{attribute 'global_init_slot' := '40510'}
VAR_GLOBAL
  LblPlt_Facade                                            :FB_BA_Label:=( sObjName:='FAS', sDescr:='Fassade');
  LblPlt_Natural_smoke_extraction                          :FB_BA_Label:=( sObjName:='NRA', sDescr:='Natürlicher Rauchabzug');
  LblPlt_Doors_gates_sluices                               :FB_BA_Label:=( sObjName:='TUE', sDescr:='Türen, Tore, Schleusen');
  LblPlt_Smoke_and_heat_extraction_system                  :FB_BA_Label:=( sObjName:='RWA', sDescr:='Rauch- und Wärmeabzugsanlage');
  LblPlt_Sunlight_protection                               :FB_BA_Label:=( sObjName:='SON', sDescr:='Sonnenschutzanlage');
// 411 Abwasseranlagen
  LblPlt_Separator_facility                                :FB_BA_Label:=( sObjName:='ABS', sDescr:='Abscheideranlage');
  LblPlt_Lifting_system                                    :FB_BA_Label:=( sObjName:='HBA', sDescr:='Hebeanlage');
  LblPlt_Neutralisation_plant                              :FB_BA_Label:=( sObjName:='NEU', sDescr:='Neutralisationsanlage');
// 412 Wasseranlagen
  LblPlt_Trace_heating                                     :FB_BA_Label:=( sObjName:='BGH', sDescr:='Begleitheizung');
  LblPlt_Process_water                                     :FB_BA_Label:=( sObjName:='BTW', sDescr:='Betriebswasser');
  LblPlt_Well_water                                        :FB_BA_Label:=( sObjName:='BWA', sDescr:='Brunnenwasser');
  LblPlt_Dispensing_installation                           :FB_BA_Label:=( sObjName:='DOS', sDescr:='Dosieranlage');
  LblPlt_Pressure_booster_system                           :FB_BA_Label:=( sObjName:='DEA', sDescr:='Druckerhöhungsanlage');
  LblPlt_Softening_unit                                    :FB_BA_Label:=( sObjName:='EHA', sDescr:='Enthärtungsanlage');
// Trinkwasser
  LblPlt_Drinking_water_heating_system                     :FB_BA_Label:=( sObjName:='TWE', sDescr:='Trinkwassererwärmungsanlage');
  LblPlt_Reverse_osmosis_system                            :FB_BA_Label:=( sObjName:='UKO', sDescr:='Umkehrosmoseanlage');
  LblPlt_Desalination_plant                                :FB_BA_Label:=( sObjName:='VEA', sDescr:='Vollentsalzungsanlage');
// 421 Wärmeerzeugungsanlagen
  LblPlt_BHKW                                              :FB_BA_Label:=( sObjName:='BHK', sDescr:='BHKW');
  LblPlt_Electric_heating                                  :FB_BA_Label:=( sObjName:='EHZ', sDescr:='Elektroheizung');
  LblPlt_District_heating_transfer                         :FB_BA_Label:=( sObjName:='FWÜ', sDescr:='Fernwärmeübergabe');
// Geothermieanlage
  LblPlt_Boiler                                            :FB_BA_Label:=( sObjName:='KES', sDescr:='Kessel');
  LblPlt_Clean_steam_generation                            :FB_BA_Label:=( sObjName:='RDE', sDescr:='Reindampferzeugung');
  LblPlt_Solar_power_system                                :FB_BA_Label:=( sObjName:='SOL', sDescr:='Solaranlage');
  LblPlt_Heating_pump                                      :FB_BA_Label:=( sObjName:='WPU', sDescr:='Wärmepumpe');
// 422 Wärmeverteilnetze
  LblPlt_Pressure_maintenance                              :FB_BA_Label:=( sObjName:='DHG', sDescr:='Druckhaltung');
  LblPlt_Heating_circuit                                   :FB_BA_Label:=( sObjName:='HZK', sDescr:='Heizkreis');
  LblPlt_Heating                                           :FB_BA_Label:=( sObjName:='HZG', sDescr:='Heizung');
  LblPlt_Back_feed_system                                  :FB_BA_Label:=( sObjName:='NSA', sDescr:='Nachspeiseanlage');
  LblPlt_Buffer                                            :FB_BA_Label:=( sObjName:='PFS', sDescr:='Pufferspeicher');
  LblPlt_Heat_distribution_network                         :FB_BA_Label:=( sObjName:='WVN', sDescr:='Wärmeverteilnetz');
  LblPlt_Heat_exchanger                                    :FB_BA_Label:=( sObjName:='WTR', sDescr:='Wärmeüberträger');
// 423 Raumheizflächen
  LblPlt_Concrete_core_activation                          :FB_BA_Label:=( sObjName:='BKA', sDescr:='Betonkernaktivierung');
  LblPlt_Overhead_heating                                  :FB_BA_Label:=( sObjName:='DHZ', sDescr:='Deckenheizung');
  LblPlt_Ceiling_radiator_panels                           :FB_BA_Label:=( sObjName:='DSP', sDescr:='Deckenstrahlplatten');
  LblPlt_Facade_heating                                    :FB_BA_Label:=( sObjName:='FAH', sDescr:='Fassadenheizung');
  LblPlt_Panel_heating                                     :FB_BA_Label:=( sObjName:='FLH', sDescr:='Flächenheizung');
  LblPlt_Underfloor_heating                                :FB_BA_Label:=( sObjName:='FBH', sDescr:='Fußbodenheizung');
  LblPlt_Heated_chilled_ceiling                            :FB_BA_Label:=( sObjName:='HKD', sDescr:='Heiz-/Kühldecke');
  LblPlt_Static_heating                                    :FB_BA_Label:=( sObjName:='STH', sDescr:='Statische Heizung');
// 430 Lufttechnische Anlagen
  LblPlt_Extract_air_system                                :FB_BA_Label:=( sObjName:='ABA', sDescr:='Abluftanlage');
  LblPlt_Roof_air_heater                                   :FB_BA_Label:=( sObjName:='DLH', sDescr:='Deckenlufterhitzer');
  LblPlt_Circulatory_system                                :FB_BA_Label:=( sObjName:='KVS', sDescr:='Kreislaufverbundsystem');
  LblPlt_Air_processing_unit                               :FB_BA_Label:=( sObjName:='LAZ', sDescr:='Luftaufbereitungszentrale');
  LblPlt_Mechanical_smoke_extraction_system                :FB_BA_Label:=( sObjName:='MRA', sDescr:='Maschinelle Rauchabzugsanlage');
  LblPlt_Smoke_pressure_system                             :FB_BA_Label:=( sObjName:='RDA', sDescr:='Rauchdruckanlage');
  LblPlt_Air_handling_unit                                 :FB_BA_Label:=( sObjName:='RLT', sDescr:='Raumlufttechnik');
  LblPlt_Partial_air_conditioning_system                   :FB_BA_Label:=( sObjName:='TKA', sDescr:='Teilklimaanlage');
  LblPlt_Air_curtain_system                                :FB_BA_Label:=( sObjName:='TLS', sDescr:='Türluftschleieranlage');
  LblPlt_Recirculating_air_system                          :FB_BA_Label:=( sObjName:='ULA', sDescr:='Umluftanlage');
  LblPlt_Full_air_conditioning_system                      :FB_BA_Label:=( sObjName:='VKA', sDescr:='Vollklimaanlage');
  LblPlt_Heat_recovery_system                              :FB_BA_Label:=( sObjName:='WRG', sDescr:='Wärmerückgewinnungssystem');
  LblPlt_Intake_air_system                                 :FB_BA_Label:=( sObjName:='ZUA', sDescr:='Zuluftanlage');
  LblPlt_Smoke_extraction_system                           :FB_BA_Label:=( sObjName:='ERA', sDescr:='Entrauchungsanlage');
// 434 Kälteanlagen
  LblPlt_Remote_cooling_transfer                           :FB_BA_Label:=( sObjName:='FKÜ', sDescr:='Fernkälteübergabe');
  LblPlt_Cooling                                           :FB_BA_Label:=( sObjName:='KAE', sDescr:='Kälte');
  LblPlt_Cooling_circuit                                   :FB_BA_Label:=( sObjName:='KKR', sDescr:='Kältekreis');
  LblPlt_Cooling_distribution_network                      :FB_BA_Label:=( sObjName:='KVN', sDescr:='Kälteverteilnetz');
  LblPlt_Cold_water_generation                             :FB_BA_Label:=( sObjName:='KWE', sDescr:='Kaltwassererzeugung');
  LblPlt_Electrical_cabinet_cooling                        :FB_BA_Label:=( sObjName:='KVE', sDescr:='Kühlung Schaltschrank ');
  LblPlt_Cooling_storage                                   :FB_BA_Label:=( sObjName:='KSP', sDescr:='Kältespeicher');
  LblPlt_Chilled_ceiling                                   :FB_BA_Label:=( sObjName:='KÜD', sDescr:='Kühldecke');
  LblPlt_Re_cooling_plant                                  :FB_BA_Label:=( sObjName:='RKW', sDescr:='Rückkühlwerk');
// 441 Hoch- und Mittelspannungsanlagen
  LblPlt_Switchgear                                        :FB_BA_Label:=( sObjName:='STA', sDescr:='Schaltanlagen');
  LblPlt_Transformer                                       :FB_BA_Label:=( sObjName:='TRF', sDescr:='Transformator');
  LblPlt_Medium_voltage_system                             :FB_BA_Label:=( sObjName:='MSA', sDescr:='Mittelspannungsanlage');
  LblPlt_Compensation_system                               :FB_BA_Label:=( sObjName:='KOA', sDescr:='Kompensationsanlage');
  LblPlt_Frequency_converter_system                        :FB_BA_Label:=( sObjName:='FUA', sDescr:='Frequenzumformeranlage');
// 442 Eigenstromversorgungsanlagen
  LblPlt_Emissions_system                                  :FB_BA_Label:=( sObjName:='AGA', sDescr:='Abgasanlage');
  LblPlt_Battery_unit                                      :FB_BA_Label:=( sObjName:='BAT', sDescr:='Batterieanlage');
  LblPlt_Co_generation_unit                                :FB_BA_Label:=( sObjName:='BHK', sDescr:='Blockheizkraftwerk');
  LblPlt_Fuel_supply                                       :FB_BA_Label:=( sObjName:='BRV', sDescr:='Brennstoffversorgung');
  LblPlt_Standby_power_system                              :FB_BA_Label:=( sObjName:='ESA', sDescr:='Ersatzstromanlage');
  LblPlt_Photovoltaic_system                               :FB_BA_Label:=( sObjName:='PVA', sDescr:='Fotovoltaikanlage');
  LblPlt_Uninterruptible_power_supply                      :FB_BA_Label:=( sObjName:='USV', sDescr:='Unterbrechungsfreie Stromversorgung');
// 443 Niederspannungsschaltanlagen
  LblPlt_General_power_supply                              :FB_BA_Label:=( sObjName:='ASV', sDescr:='Allgemeine Stromversorgung');
  LblPlt_Safety_power_supply                               :FB_BA_Label:=( sObjName:='SSV', sDescr:='Sicherheitsstromversorgung');
  LblPlt_Lighting                                          :FB_BA_Label:=( sObjName:='BEL', sDescr:='Beleuchtungsanlage');
  LblPlt_Emergency_lighting                                :FB_BA_Label:=( sObjName:='SIB', sDescr:='Sicherheitsbeleuchtung');
// 451 Telekommunikationsanlagen
  LblPlt_Telecommunications_system                         :FB_BA_Label:=( sObjName:='TEL', sDescr:='Telekommunikationsanlage');
// 452 Such- und Signalanlagen
  LblPlt_Call_signalling_system                            :FB_BA_Label:=( sObjName:='LRA', sDescr:='Lichtrufanlage');
  LblPlt_Door_intercom_and_door_opener_system              :FB_BA_Label:=( sObjName:='TÜA', sDescr:='Türsprech- und -öffneranlage');
  LblPlt_Paging_system                                     :FB_BA_Label:=( sObjName:='PRA', sDescr:='Personenrufanlage');
// 453 Zeitdienstanlagen
  LblPlt_Clock_and_time_recording_system                   :FB_BA_Label:=( sObjName:='ZEA', sDescr:='Uhren- und Zeiterfassungsanlage');
// 454 Elektroakustische Anlagen
  LblPlt_Electro_acoustic_sound_systems                    :FB_BA_Label:=( sObjName:='ELA', sDescr:='Elektroakustische Anl. , Beschallung');
  LblPlt_Conference_and_interpreting_equipment             :FB_BA_Label:=( sObjName:='KDA', sDescr:='Konferenz- und Dolmetscheranlage');
  LblPlt_Intercom_system                                   :FB_BA_Label:=( sObjName:='GSA', sDescr:='Gegensprechanlage');
  LblPlt_Voice_alarm_system                                :FB_BA_Label:=( sObjName:='SAA', sDescr:='Sprachalarmierungsanlage');
  LblPlt_Intercommunication_systems                        :FB_BA_Label:=( sObjName:='WSA', sDescr:='Wechselsprechanlagen');
// 455 Fernseh- und Antennenanlagen
  LblPlt_Television_system                                 :FB_BA_Label:=( sObjName:='TVA', sDescr:='Fernsehanlage');
  LblPlt_Transmitting_and_receiving_antenna_system         :FB_BA_Label:=( sObjName:='SEA', sDescr:='Sende- und Empfangsantennenanlage');
  LblPlt_BOS_radio_system                                  :FB_BA_Label:=( sObjName:='BOS', sDescr:='BOS-Funkanlage');
// 456 Gefahrenmelde- und Alarmanlagen
  LblPlt_Fire_detection_and_alarm_systems                  :FB_BA_Label:=( sObjName:='BMA', sDescr:='Brandmeldeanlage');
  LblPlt_Carbon_monoxide_warning_system                    :FB_BA_Label:=( sObjName:='COW', sDescr:='CO-Warnanlage');
  LblPlt_Burglar_alarm_systems                             :FB_BA_Label:=( sObjName:='EMA', sDescr:='Einbruchmeldeanlage');
  LblPlt_Fire_control_panel                                :FB_BA_Label:=( sObjName:='FWT', sDescr:='Feuerwehrtableau');
  LblPlt_Escape_route_protection_system                    :FB_BA_Label:=( sObjName:='FWS', sDescr:='Fluchtwegsicherungsanlage');
  LblPlt_Hazard_detection_system                           :FB_BA_Label:=( sObjName:='GMA', sDescr:='Gefahrenmeldeanlage');
  LblPlt_Gas_warning_system                                :FB_BA_Label:=( sObjName:='GWA', sDescr:='Gaswarnanlage');
  LblPlt_Smoke_aspiration_system                           :FB_BA_Label:=( sObjName:='RAS', sDescr:='Rauchansaugsystem');
  LblPlt_Room_observation_system                           :FB_BA_Label:=( sObjName:='RBA', sDescr:='Raumbeobachtungsanlage');
  LblPlt_Robbery_alarm_system                              :FB_BA_Label:=( sObjName:='ÜFA', sDescr:='Überfallmeldeanlage');
  LblPlt_Guard_control_system                              :FB_BA_Label:=( sObjName:='WKA', sDescr:='Wächterkontrollanlage');
  LblPlt_Emergency_call_system                             :FB_BA_Label:=( sObjName:='NOT', sDescr:='Notrufanlage');
  LblPlt_Access_control_system                             :FB_BA_Label:=( sObjName:='ZKS', sDescr:='Zugangskontrollsystem');
// 457 Übertragungsnetze
  LblPlt_Networks_for_the_transmission_voice_text_etc      :FB_BA_Label:=( sObjName:='LAN', sDescr:='Netzw.  Daten, Sprache, Text etc');
// 459 Fernmelde- und informationstechnische Anlagen, Sonstiges
  LblPlt_Remote_control_systems                            :FB_BA_Label:=( sObjName:='FWA', sDescr:='Fernwirkanlagen');
  LblPlt_Parking_guidance_systems                          :FB_BA_Label:=( sObjName:='PLS', sDescr:='Parkleitsysteme');
// 460 Förderanlagen
  LblPlt_File_transportation_systems                       :FB_BA_Label:=( sObjName:='ATA', sDescr:='Aktentransportanlagen');
  LblPlt_Lift                                              :FB_BA_Label:=( sObjName:='AUF', sDescr:='Aufzug');
  LblPlt_Inspection_systems                                :FB_BA_Label:=( sObjName:='BFA', sDescr:='Befahranlagen');
  LblPlt_Moving_walkways                                   :FB_BA_Label:=( sObjName:='FST', sDescr:='Fahrsteige');
  LblPlt_Escalators                                        :FB_BA_Label:=( sObjName:='FTR', sDescr:='Fahrtreppen');
  LblPlt_External_lifts                                    :FB_BA_Label:=( sObjName:='FSA', sDescr:='Fassadenaufzüge');
  LblPlt_Baggage_conveyor_system                           :FB_BA_Label:=( sObjName:='GFA', sDescr:='Gepäckförderanlage');
  LblPlt_Pneumatic_delivery_systems                        :FB_BA_Label:=( sObjName:='RPA', sDescr:='Rohrpostanlagen');
  LblPlt_Goods_transportation_facilities                   :FB_BA_Label:=( sObjName:='WTA', sDescr:='Warentransportanlagen');
// 470 Nutzerspezifische Anlagen
// 471 Küchentechnische Anlagen
  LblPlt_Small_refrigeration_unit                          :FB_BA_Label:=( sObjName:='KLK', sDescr:='Kleinkälteanlage');
// 472 Wäscherei- und Reinigungsanlagen
  LblPlt_Disinfection_unit                                 :FB_BA_Label:=( sObjName:='DES', sDescr:='Desinfektionsanlage');
  LblPlt_Cleaning_unit                                     :FB_BA_Label:=( sObjName:='REA', sDescr:='Reinigungsanlage');
  LblPlt_Sterilisation_systems                             :FB_BA_Label:=( sObjName:='STR', sDescr:='Sterilisationseinrichtungen');
  LblPlt_Water_treatment_system                            :FB_BA_Label:=( sObjName:='WAA', sDescr:='Wasseraufbereitungsanlage');
  LblPlt_Laundry_system                                    :FB_BA_Label:=( sObjName:='WÄA', sDescr:='Wäschereianlage');
// 473 Medienversorgungsanlagen
  LblPlt_Compressed_air_supply_system                      :FB_BA_Label:=( sObjName:='DRL', sDescr:='Druckluftversorgungsanlage');
  LblPlt_Pressure_regulator_unit                           :FB_BA_Label:=( sObjName:='DRA', sDescr:='Druckregelanlage');
  LblPlt_Media_supply_system                               :FB_BA_Label:=( sObjName:='MVA', sDescr:='Medienversorgungsanlage');
  LblPlt_Medical_and_technical_gases                       :FB_BA_Label:=( sObjName:='MTG', sDescr:='Medizinische und technische Gase');
  LblPlt_Vacuum_unit                                       :FB_BA_Label:=( sObjName:='VAK', sDescr:='Vakuumanlage');
// 474 Medizin- und labortechnische Anlagen
  LblPlt_Medical_technical_plant                           :FB_BA_Label:=( sObjName:='MED', sDescr:='Medizintechnische Anlagen');
  LblPlt_Medical_gas_supply                                :FB_BA_Label:=( sObjName:='MGV', sDescr:='Medizinische Gasversorgung');
  LblPlt_Laboratory_equipment                              :FB_BA_Label:=( sObjName:='LAB', sDescr:='Labortechnische Anlagen (allgemein)');
// 475 Feuerlöschanlagen
  LblPlt_Fire_extinguisher                                 :FB_BA_Label:=( sObjName:='FLA', sDescr:='Feuerlöschanlage');
  LblPlt_Gas_extinguishing_system                          :FB_BA_Label:=( sObjName:='GLA', sDescr:='Gaslöschanlage');
  LblPlt_Fire_extinguishing_system                         :FB_BA_Label:=( sObjName:='LÖS', sDescr:='Löschanlage (allgemein)');
  LblPlt_Mist_extinguishing_system                         :FB_BA_Label:=( sObjName:='NLA', sDescr:='Nebellöschanlage');
  LblPlt_NOX_system                                        :FB_BA_Label:=( sObjName:='NOX', sDescr:='NOX-Anlage');
  LblPlt_Sprinkler_system                                  :FB_BA_Label:=( sObjName:='SPR', sDescr:='Sprinkleranlage');
  LblPlt_Wall_hydrant_system                               :FB_BA_Label:=( sObjName:='WHA', sDescr:='Wandhydrantenanlage');
// 478 Entsorgungsanlagen
  LblPlt_Waste_disposal_system                             :FB_BA_Label:=( sObjName:='AEA', sDescr:='Abfallentsorgungsanlage');
  LblPlt_Media_disposal_system                             :FB_BA_Label:=( sObjName:='MEA', sDescr:='Medienentsorgungsanlage');
  LblPlt_Vacuum_cleaning_systems                           :FB_BA_Label:=( sObjName:='SSA', sDescr:='Staubsauganlagen');
// 480 Gebäudeautomation
  LblPlt_Automation_control_equipment                      :FB_BA_Label:=( sObjName:='ASP', sDescr:='Automationsschwerpunkt');
  LblPlt_Weather_station                                   :FB_BA_Label:=( sObjName:='WET', sDescr:='Wetterstation');
  LblPlt_Weather_data                                      :FB_BA_Label:=( sObjName:='WED', sDescr:='Wetterdaten');
  LblPlt_Management_and_operating_equipment                :FB_BA_Label:=( sObjName:='MBE', sDescr:='Management- und Bedieneinrichtungen');
  LblPlt_Room_automation                                   :FB_BA_Label:=( sObjName:='RAU', sDescr:='Raumautomation');
  LblPlt_Room_automation_system_distributor                :FB_BA_Label:=( sObjName:='RAV', sDescr:='Raumautomation-Systemverteiler');
  LblPlt_Control_cabinet                                   :FB_BA_Label:=( sObjName:='SSK', sDescr:='Schaltschrank');
  LblPlt_Settings                                          :FB_BA_Label:=( sObjName:='ALP', sDescr:='Anlagenparameter');
  LblPlt_EventGroups                                       :FB_BA_Label:=( sObjName:='ERG', sDescr:='Meldeklassen');
  LblPlt_Global_building_data                              :FB_BA_Label:=( sObjName:='GGL', sDescr:='Globale Gebäudedaten');
// 540 Technische Anlagen in Außenanlagen
  LblPlt_Rainwater_retention_basin                         :FB_BA_Label:=( sObjName:='RRB', sDescr:='Regenrückhaltebecken');
  LblPlt_Cistern_system                                    :FB_BA_Label:=( sObjName:='ZTA', sDescr:='Zisternenanlage');
END_VAR

// ---- Templates/GVLs/Language/German/TxtEvent_DE.TcGVL
{region '#Template'}
	{attribute 'Version' := '5.1.0.0'}
	{attribute 'Tags' := '"LCID": "1031", "Text": "GVL, Property, Event, Event Message Text, Active Text, Inactive Text"'}
	{attribute 'Tags' := '"LCID": "1033", "Text": "GVL, Property, Event, Event Message Text, Active Text, Inactive Text"'}
	{attribute 'Description' := '"LCID": "1031", "Text": "Textliste Properties Event Message Text, Active Text, Inactive Text"'}
	{attribute 'Description' := '"LCID": "1033", "Text": "Text list Properties Event Message Text, Active Text, Inactive Text"'}
{endregion}

{attribute 'global_init_slot' := '40510'}
VAR_GLOBAL
  txtEvent_No                                                :T_BA_StateText:='Nein';
  txtEvent_Yes                                               :T_BA_StateText:='Ja';
  txtEvent_Auto                                              :T_BA_StateText:='Automatik';
  txtEvent_Manual                                            :T_BA_StateText:='Hand';
  txtEvent_Off                                               :T_BA_StateText:='Aus';
  txtEvent_On                                                :T_BA_StateText:='Ein';
  txtEvent_Opened                                            :T_BA_StateText:='Geöffnet';
  txtEvent_Closed                                            :T_BA_StateText:='Geschlossen';
  txtEvent_Open                                              :T_BA_StateText:='Auf';
  txtEvent_Close                                             :T_BA_StateText:='Zu';
  txtEvent_Step1                                             :T_BA_StateText:='Stufe 1 ';
  txtEvent_Step2                                             :T_BA_StateText:='Stufe 2';
  txtEvent_Step3                                             :T_BA_StateText:='Stufe 3';
  txtEvent_Step4                                             :T_BA_StateText:='Stufe 4';
  txtEvent_Step5                                             :T_BA_StateText:='Stufe 5';
  txtEvent_Step6                                             :T_BA_StateText:='Stufe 6';
  txtEvent_Step7                                             :T_BA_StateText:='Stufe 7';
  txtEvent_Step8                                             :T_BA_StateText:='Stufe 8';
  txtEvent_Released                                          :T_BA_StateText:='Freigegeben';
  txtEvent_Inactive                                          :T_BA_StateText:='Inaktiv';
  txtEvent_Active                                            :T_BA_StateText:='Aktiv';
  txtEvent_Normal                                            :T_BA_StateText:='Normal';
  txtEvent_Offnormal                                         :T_BA_StateText:='Unnormal';
  txtEvent_Alert                                             :T_BA_StateText:='Alarm';
  txtEvent_Disturb                                           :T_BA_StateText:='Störung';
  txtEvent_Error                                             :T_BA_StateText:='Fehler ';
  txtEvent_Triggered                                         :T_BA_StateText:='Ausgelöst';
  txtEvent_Maintenace                                        :T_BA_StateText:='Wartung';
  txtEvent_Exceeded                                          :T_BA_StateText:='Überschritten';
  txtEvent_Monitoring                                        :T_BA_StateText:='Überwachung';
  txtEvent_Protection                                        :T_BA_StateText:='Schutzbetrieb';
  txtEvent_Economy                                           :T_BA_StateText:='Economy';
  txtEvent_PreComfort                                        :T_BA_StateText:='Pre-Comfort';
  txtEvent_Comfort                                           :T_BA_StateText:='Comfort';
  txtEvent_Reached                                           :T_BA_StateText:='erreicht';
  txtEvent_NotReached                                        :T_BA_StateText:='nicht erreicht';
  txtEvent_None                                              :T_BA_StateText:='""';
  txtEvent_EmergencyStop                                     :T_BA_StateText:='Notaus';
  txtEvent_Frost                                             :T_BA_StateText:='Frost';
  txtEvent_SmokeExtraction_P                                 :T_BA_StateText:='Entrauchung mit Zu- und Abluft';
  txtEvent_SmokeExtractionSupplyAir                          :T_BA_StateText:='Entrauchung Zuluft';
  txtEvent_SmokeExtractionExtractAir                         :T_BA_StateText:='Entrauchung Abluft';
  txtEvent_CoolDownProtection                                :T_BA_StateText:='Auskühlschutz';
  txtEvent_OverHeatingProtection                             :T_BA_StateText:='Überhitzungsschutz';
  txtEvent_Fire                                              :T_BA_StateText:='Brandalarm';
  txtEvent_NightCooling                                      :T_BA_StateText:='Nachtkühlung';
  txtEvent_ForcedVentilation                                 :T_BA_StateText:='Zwangsbelüftung';
  txtEvent_CentralSwitchOff                                  :T_BA_StateText:='Zentralaus';
  txtEvent_Locked                                            :T_BA_StateText:='verriegelt';
  txtEvent_Contaminated                                      :T_BA_StateText:='verschmutzt';
  txtEvent_Stop                                              :T_BA_StateText:='Stop';
  txtEvent_Critical                                          :T_BA_StateText:='kritisch';
  txtEvent_CriticalOn                                        :T_BA_StateText:='kritisch ein';
  txtEvent_CriticalOff                                       :T_BA_StateText:='kritisch aus';
  txtEvent_UnCiritical                                       :T_BA_StateText:='unkritisch';
  txtEvent_LifeSafetyOn                                      :T_BA_StateText:='Lebensgefahr ein';
  txtEvent_LifeSafetyOff                                     :T_BA_StateText:='Lebensgefahr aus';
  txtEvent_Average                                           :T_BA_StateText:='Mittelwert';
  txtEvent_HeatCool                                          :T_BA_StateText:='Heiz/Kühl';
  txtEvent_AverageHeatCool                                   :T_BA_StateText:='Mittelwert Heizen/Kühlen';
  txtEvent_Direction                                         :T_BA_StateText:='Wirksinn';
  txtEvent_Default                                           :T_BA_StateText:='Standard';
  txtEvent_Cleaning                                          :T_BA_StateText:='Gebaeudereinigung';
  txtEvent_Nightwatch                                        :T_BA_StateText:='Nachtwaechter';
  txtEvent_SupplyAirTControlReheater                         :T_BA_StateText:='Zulufttemperaturregelung Nacherhitzer';
  txtEvent_SupplyAirTControlPreheater                        :T_BA_StateText:='Zulufttemperaturregelung Vorerhitzer';
  txtEvent_SupplyAirTControlERC                              :T_BA_StateText:='Zulufttemperaturregelung WRG';
  txtEvent_SupplyAirTControlMix                              :T_BA_StateText:='Zulufttemperaturregelung Mischluft';
  txtEvent_SupplyAirTControlCooler                           :T_BA_StateText:='Zulufttemperaturregelung Kühler';
  txtEvent_SupplyAirXControlCooler                           :T_BA_StateText:='Zuluftfeuchtereglung Kühler';
  txtEvent_SupplyAirXControlHumf                             :T_BA_StateText:='Zuluftfeuchtereglung Befeuchter';
  txtEvent_PreRinse                                          :T_BA_StateText:='Vorspülen';
  txtEvent_DamperOpen                                        :T_BA_StateText:='Klappen Auf';
  txtEvent_SupplyAirFan                                      :T_BA_StateText:='Zuluft Ventilator';
  txtEvent_ExtractAirFan                                     :T_BA_StateText:='Abluft Ventilator';
  txtEvent_EnableTemperatureControl                          :T_BA_StateText:='Freigabe Temperatur Regelung';
  txtEvent_EnableTemperatureSequenceLink                     :T_BA_StateText:='Freigabe Temperatur Sequenz Steuerung';
  txtEvent_EnableHumidityControl                             :T_BA_StateText:='Freigabe Feuchte Regelung';
  txtEvent_EnableHumiditySequenceLink                        :T_BA_StateText:='Freigabe Feuchte Sequenz Steuerung';
  txtEvent_ReleaseLimitMonitoring                            :T_BA_StateText:='Freigabe Grenzwertüberwachung';
  txtEvent_Reheater                                          :T_BA_StateText:='Nacherhitzer';
  txtEvent_Preheater                                         :T_BA_StateText:='Vorerhitzer';
  txtEvent_MixedAir                                          :T_BA_StateText:='Mischluft';
  txtEvent_EnergyRecovery                                    :T_BA_StateText:='Energierückgewinnung';
  txtEvent_Cooler                                            :T_BA_StateText:='Kühler';
  txtEvent_Humidifier                                        :T_BA_StateText:='Befeuchter';
  txtEvent_Dehumidifier                                      :T_BA_StateText:='Entfeuchter';
  txtEvent_DamperExhaustAir                                  :T_BA_StateText:='Fortluftklappe';
  txtEvent_DamperOutsideAir                                  :T_BA_StateText:='Aussenluftklappe';
  txtEvent_Occupied                                          :T_BA_StateText:='Belegt';
  txtEvent_NotOccupied                                       :T_BA_StateText:='Nicht belegt';
  txtEvent_Storm                                             :T_BA_StateText:='Sturmalarm';
  txtEvent_Ice                                               :T_BA_StateText:='Vereisung';
  txtEvent_CommError                                         :T_BA_StateText:='Kommunikationsfehler';
  txtEvent_Burglary                                          :T_BA_StateText:='Einbruch';
  txtEvent_Maintenance                                       :T_BA_StateText:='Wartung';
  txtEvent_Referencing                                       :T_BA_StateText:='Referenzieren';
  txtEvent_ManualActuator                                    :T_BA_StateText:='Hand Einzel';
  txtEvent_ManualGroup                                       :T_BA_StateText:='Hand Gruppe';
  txtEvent_AllDown                                           :T_BA_StateText:='Alle herab';
  txtEvent_AllUp                                             :T_BA_StateText:='Alle herauf';
  txtEvent_Scene1                                            :T_BA_StateText:='Szene 1';
  txtEvent_FacadeThermoAutomatic                             :T_BA_StateText:='Fassaden-Thermoautomatik';
  txtEvent_FacadeTwilightAutomatic                           :T_BA_StateText:='Fassaden-Dämmerungsautomatik';
  txtEvent_ParkPosition                                      :T_BA_StateText:='Parkposition';
  txtEvent_Scene2                                            :T_BA_StateText:='Szene 2';
  txtEvent_Scene3                                            :T_BA_StateText:='Szene 3';
  txtEvent_SunProtection                                     :T_BA_StateText:='Sonnenschutz';
  txtEvent_GroupThermoAuto                                   :T_BA_StateText:='Thermoautomatik';
  txtEvent_GroupTwiLightAuto                                 :T_BA_StateText:='Dämmerungsautomatik';
  txtEvent_UserDefined1                                      :T_BA_StateText:='Benutzerdefiniert 1';
  txtEvent_UserDefined2                                      :T_BA_StateText:='Benutzerdefiniert 2';
END_VAR

// ---- Templates/GVLs/Language/German/TxtPlant_DE.TcGVL
{region '#Template'}
	{attribute 'Version' := '5.0.0.0'}
	{attribute 'Tags' := '"LCID": "1031", "Text": "GVL, DPAD, Plants, ObjectName, Description"'}
	{attribute 'Tags' := '"LCID": "1033", "Text": "GVL, DPAD, Plants, ObjectName, Description"'}
	{attribute 'Description' := '"LCID": "1031", "Text": "Textliste Anlagen"'}
	{attribute 'Description' := '"LCID": "1033", "Text": "Text list plants"'}
{endregion}

{attribute 'global_init_slot' := '40510'}
VAR_GLOBAL
  TxTPlant_Facade_sObjectName                                            :T_BA_StateText:='FAS';
  TxTPlant_Facade_sDescription                                            :T_BA_StateText:='Fassade';
  TxTPlant_Natural_smoke_extraction_sObjectName                          :T_BA_StateText:='NRA';
  TxTPlant_Natural_smoke_extraction_sDescription                          :T_BA_StateText:='Natürlicher Rauchabzug';
  TxTPlant_Doors_gates_sluices_sObjectName                               :T_BA_StateText:='TUE';
  TxTPlant_Doors_gates_sluices_sDescription                               :T_BA_StateText:='Türen, Tore, Schleusen';
  TxTPlant_Smoke_and_heat_extraction_system_sObjectName                  :T_BA_StateText:='RWA';
  TxTPlant_Smoke_and_heat_extraction_system_sDescription                  :T_BA_StateText:='Rauch- und Wärmeabzugsanlage';
  TxTPlant_Sunlight_protection_sObjectName                               :T_BA_StateText:='SON';
  TxTPlant_Sunlight_protection_sDescription                               :T_BA_StateText:='Sonnenschutzanlage';
// 411 Abwasseranlagen
  TxTPlant_Separator_facility_sObjectName                                :T_BA_StateText:='ABS';
  TxTPlant_Separator_facility_sDescription                                :T_BA_StateText:='Abscheideranlage';
  TxTPlant_Lifting_system_sObjectName                                    :T_BA_StateText:='HBA';
  TxTPlant_Lifting_system_sDescription                                    :T_BA_StateText:='Hebeanlage';
  TxTPlant_Neutralisation_plant_sObjectName                              :T_BA_StateText:='NEU';
  TxTPlant_Neutralisation_plant_sDescription                              :T_BA_StateText:='Neutralisationsanlage';
// 412 Wasseranlagen
  TxTPlant_Trace_heating_sObjectName                                     :T_BA_StateText:='BGH';
  TxTPlant_Trace_heating_sDescription                                     :T_BA_StateText:='Begleitheizung';
  TxTPlant_Process_water_sObjectName                                     :T_BA_StateText:='BTW';
  TxTPlant_Process_water_sDescription                                     :T_BA_StateText:='Betriebswasser';
  TxTPlant_Well_water_sObjectName                                        :T_BA_StateText:='BWA';
  TxTPlant_Well_water_sDescription                                        :T_BA_StateText:='Brunnenwasser';
  TxTPlant_Dispensing_installation_sObjectName                           :T_BA_StateText:='DOS';
  TxTPlant_Dispensing_installation_sDescription                           :T_BA_StateText:='Dosieranlage';
  TxTPlant_Pressure_booster_system_sObjectName                           :T_BA_StateText:='DEA';
  TxTPlant_Pressure_booster_system_sDescription                           :T_BA_StateText:='Druckerhöhungsanlage';
  TxTPlant_Softening_unit_sObjectName                                    :T_BA_StateText:='EHA';
  TxTPlant_Softening_unit_sDescription                                    :T_BA_StateText:='Enthärtungsanlage';
// Trinkwasser
  TxTPlant_Drinking_water_heating_system_sObjectName                     :T_BA_StateText:='TWE';
  TxTPlant_Drinking_water_heating_system_sDescription                     :T_BA_StateText:='Trinkwassererwärmungsanlage';
  TxTPlant_Reverse_osmosis_system_sObjectName                            :T_BA_StateText:='UKO';
  TxTPlant_Reverse_osmosis_system_sDescription                            :T_BA_StateText:='Umkehrosmoseanlage';
  TxTPlant_Desalination_plant_sObjectName                                :T_BA_StateText:='VEA';
  TxTPlant_Desalination_plant_sDescription                                :T_BA_StateText:='Vollentsalzungsanlage';
// 421 Wärmeerzeugungsanlagen
  TxTPlant_BHKW_sObjectName                                              :T_BA_StateText:='BHK';
  TxTPlant_BHKW_sDescription                                              :T_BA_StateText:='BHKW';
  TxTPlant_Electric_heating_sObjectName                                  :T_BA_StateText:='EHZ';
  TxTPlant_Electric_heating_sDescription                                  :T_BA_StateText:='Elektroheizung';
  TxTPlant_District_heating_transfer_sObjectName                         :T_BA_StateText:='FWÜ';
  TxTPlant_District_heating_transfer_sDescription                         :T_BA_StateText:='Fernwärmeübergabe';
// Geothermieanlage
  TxTPlant_Boiler_sObjectName                                            :T_BA_StateText:='KES';
  TxTPlant_Boiler_sDescription                                            :T_BA_StateText:='Kessel';
  TxTPlant_Clean_steam_generation_sObjectName                            :T_BA_StateText:='RDE';
  TxTPlant_Clean_steam_generation_sDescription                            :T_BA_StateText:='Reindampferzeugung';
  TxTPlant_Solar_power_system_sObjectName                                :T_BA_StateText:='SOL';
  TxTPlant_Solar_power_system_sDescription                                :T_BA_StateText:='Solaranlage';
  TxTPlant_Heating_pump_sObjectName                                      :T_BA_StateText:='WPU';
  TxTPlant_Heating_pump_sDescription                                      :T_BA_StateText:='Wärmepumpe';
// 422 Wärmeverteilnetze
  TxTPlant_Pressure_maintenance_sObjectName                              :T_BA_StateText:='DHG';
  TxTPlant_Pressure_maintenance_sDescription                              :T_BA_StateText:='Druckhaltung';
  TxTPlant_Heating_circuit_sObjectName                                   :T_BA_StateText:='HZK';
  TxTPlant_Heating_circuit_sDescription                                   :T_BA_StateText:='Heizkreis';
  TxTPlant_Heating_sObjectName                                           :T_BA_StateText:='HZG';
  TxTPlant_Heating_sDescription                                           :T_BA_StateText:='Heizung';
  TxTPlant_Back_feed_system_sObjectName                                  :T_BA_StateText:='NSA';
  TxTPlant_Back_feed_system_sDescription                                  :T_BA_StateText:='Nachspeiseanlage';
  TxTPlant_Buffer_sObjectName                                            :T_BA_StateText:='PFS';
  TxTPlant_Buffer_sDescription                                            :T_BA_StateText:='Pufferspeicher';
  TxTPlant_Heat_distribution_network_sObjectName                         :T_BA_StateText:='WVN';
  TxTPlant_Heat_distribution_network_sDescription                         :T_BA_StateText:='Wärmeverteilnetz';
  TxTPlant_Heat_exchanger_sObjectName                                    :T_BA_StateText:='WTR';
  TxTPlant_Heat_exchanger_sDescription                                    :T_BA_StateText:='Wärmeüberträger';
// 423 Raumheizflächen
  TxTPlant_Concrete_core_activation_sObjectName                          :T_BA_StateText:='BKA';
  TxTPlant_Concrete_core_activation_sDescription                          :T_BA_StateText:='Betonkernaktivierung';
  TxTPlant_Overhead_heating_sObjectName                                  :T_BA_StateText:='DHZ';
  TxTPlant_Overhead_heating_sDescription                                  :T_BA_StateText:='Deckenheizung';
  TxTPlant_Ceiling_radiator_panels_sObjectName                           :T_BA_StateText:='DSP';
  TxTPlant_Ceiling_radiator_panels_sDescription                           :T_BA_StateText:='Deckenstrahlplatten';
  TxTPlant_Facade_heating_sObjectName                                    :T_BA_StateText:='FAH';
  TxTPlant_Facade_heating_sDescription                                    :T_BA_StateText:='Fassadenheizung';
  TxTPlant_Panel_heating_sObjectName                                     :T_BA_StateText:='FLH';
  TxTPlant_Panel_heating_sDescription                                     :T_BA_StateText:='Flächenheizung';
  TxTPlant_Underfloor_heating_sObjectName                                :T_BA_StateText:='FBH';
  TxTPlant_Underfloor_heating_sDescription                                :T_BA_StateText:='Fußbodenheizung';
  TxTPlant_Heated_chilled_ceiling_sObjectName                            :T_BA_StateText:='HKD';
  TxTPlant_Heated_chilled_ceiling_sDescription                            :T_BA_StateText:='Heiz-/Kühldecke';
  TxTPlant_Static_heating_sObjectName                                    :T_BA_StateText:='STH';
  TxTPlant_Static_heating_sDescription                                    :T_BA_StateText:='Statische Heizung';
// 430 Lufttechnische Anlagen
  TxTPlant_Extract_air_system_sObjectName                                :T_BA_StateText:='ABA';
  TxTPlant_Extract_air_system_sDescription                                :T_BA_StateText:='Abluftanlage';
  TxTPlant_Roof_air_heater_sObjectName                                   :T_BA_StateText:='DLH';
  TxTPlant_Roof_air_heater_sDescription                                   :T_BA_StateText:='Deckenlufterhitzer';
  TxTPlant_Circulatory_system_sObjectName                                :T_BA_StateText:='KVS';
  TxTPlant_Circulatory_system_sDescription                                :T_BA_StateText:='Kreislaufverbundsystem';
  TxTPlant_Air_processing_unit_sObjectName                               :T_BA_StateText:='LAZ';
  TxTPlant_Air_processing_unit_sDescription                               :T_BA_StateText:='Luftaufbereitungszentrale';
  TxTPlant_Mechanical_smoke_extraction_system_sObjectName                :T_BA_StateText:='MRA';
  TxTPlant_Mechanical_smoke_extraction_system_sDescription                :T_BA_StateText:='Maschinelle Rauchabzugsanlage';
  TxTPlant_Smoke_pressure_system_sObjectName                             :T_BA_StateText:='RDA';
  TxTPlant_Smoke_pressure_system_sDescription                             :T_BA_StateText:='Rauchdruckanlage';
  TxTPlant_Air_handling_unit_sObjectName                                 :T_BA_StateText:='RLT';
  TxTPlant_Air_handling_unit_sDescription                                 :T_BA_StateText:='Raumlufttechnik';
  TxTPlant_Partial_air_conditioning_system_sObjectName                   :T_BA_StateText:='TKA';
  TxTPlant_Partial_air_conditioning_system_sDescription                   :T_BA_StateText:='Teilklimaanlage';
  TxTPlant_Air_curtain_system_sObjectName                                :T_BA_StateText:='TLS';
  TxTPlant_Air_curtain_system_sDescription                                :T_BA_StateText:='Türluftschleieranlage';
  TxTPlant_Recirculating_air_system_sObjectName                          :T_BA_StateText:='ULA';
  TxTPlant_Recirculating_air_system_sDescription                          :T_BA_StateText:='Umluftanlage';
  TxTPlant_Full_air_conditioning_system_sObjectName                      :T_BA_StateText:='VKA';
  TxTPlant_Full_air_conditioning_system_sDescription                      :T_BA_StateText:='Vollklimaanlage';
  TxTPlant_Heat_recovery_system_sObjectName                              :T_BA_StateText:='WRG';
  TxTPlant_Heat_recovery_system_sDescription                              :T_BA_StateText:='Wärmerückgewinnungssystem';
  TxTPlant_Intake_air_system_sObjectName                                 :T_BA_StateText:='ZUA';
  TxTPlant_Intake_air_system_sDescription                                 :T_BA_StateText:='Zuluftanlage';
  TxTPlant_Smoke_extraction_system_sObjectName                           :T_BA_StateText:='ERA';
  TxTPlant_Smoke_extraction_system_sDescription                           :T_BA_StateText:='Entrauchungsanlage';
// 434 Kälteanlagen
  TxTPlant_Remote_cooling_transfer_sObjectName                           :T_BA_StateText:='FKÜ';
  TxTPlant_Remote_cooling_transfer_sDescription                           :T_BA_StateText:='Fernkälteübergabe';
  TxTPlant_Cooling_sObjectName                                           :T_BA_StateText:='KAE';
  TxTPlant_Cooling_sDescription                                           :T_BA_StateText:='Kälte';
  TxTPlant_Cooling_circuit_sObjectName                                   :T_BA_StateText:='KKR';
  TxTPlant_Cooling_circuit_sDescription                                   :T_BA_StateText:='Kältekreis';
  TxTPlant_Cooling_distribution_network_sObjectName                      :T_BA_StateText:='KVN';
  TxTPlant_Cooling_distribution_network_sDescription                      :T_BA_StateText:='Kälteverteilnetz';
  TxTPlant_Cold_water_generation_sObjectName                             :T_BA_StateText:='KWE';
  TxTPlant_Cold_water_generation_sDescription                             :T_BA_StateText:='Kaltwassererzeugung';
  TxTPlant_Electrical_cabinet_cooling_sObjectName                        :T_BA_StateText:='KVE';
  TxTPlant_Electrical_cabinet_cooling_sDescription                        :T_BA_StateText:='Kühlung Schaltschrank ';
  TxTPlant_Cooling_storage_sObjectName                                   :T_BA_StateText:='KSP';
  TxTPlant_Cooling_storage_sDescription                                   :T_BA_StateText:='Kältespeicher';
  TxTPlant_Chilled_ceiling_sObjectName                                   :T_BA_StateText:='KÜD';
  TxTPlant_Chilled_ceiling_sDescription                                   :T_BA_StateText:='Kühldecke';
  TxTPlant_Re_cooling_plant_sObjectName                                  :T_BA_StateText:='RKW';
  TxTPlant_Re_cooling_plant_sDescription                                  :T_BA_StateText:='Rückkühlwerk';
// 441 Hoch- und Mittelspannungsanlagen
  TxTPlant_Switchgear_sObjectName                                        :T_BA_StateText:='STA';
  TxTPlant_Switchgear_sDescription                                        :T_BA_StateText:='Schaltanlagen';
  TxTPlant_Transformer_sObjectName                                       :T_BA_StateText:='TRF';
  TxTPlant_Transformer_sDescription                                       :T_BA_StateText:='Transformator';
  TxTPlant_Medium_voltage_system_sObjectName                             :T_BA_StateText:='MSA';
  TxTPlant_Medium_voltage_system_sDescription                             :T_BA_StateText:='Mittelspannungsanlage';
  TxTPlant_Compensation_system_sObjectName                               :T_BA_StateText:='KOA';
  TxTPlant_Compensation_system_sDescription                               :T_BA_StateText:='Kompensationsanlage';
  TxTPlant_Frequency_converter_system_sObjectName                        :T_BA_StateText:='FUA';
  TxTPlant_Frequency_converter_system_sDescription                        :T_BA_StateText:='Frequenzumformeranlage';
// 442 Eigenstromversorgungsanlagen
  TxTPlant_Emissions_system_sObjectName                                  :T_BA_StateText:='AGA';
  TxTPlant_Emissions_system_sDescription                                  :T_BA_StateText:='Abgasanlage';
  TxTPlant_Battery_unit_sObjectName                                      :T_BA_StateText:='BAT';
  TxTPlant_Battery_unit_sDescription                                      :T_BA_StateText:='Batterieanlage';
  TxTPlant_Co_generation_unit_sObjectName                                :T_BA_StateText:='BHK';
  TxTPlant_Co_generation_unit_sDescription                                :T_BA_StateText:='Blockheizkraftwerk';
  TxTPlant_Fuel_supply_sObjectName                                       :T_BA_StateText:='BRV';
  TxTPlant_Fuel_supply_sDescription                                       :T_BA_StateText:='Brennstoffversorgung';
  TxTPlant_Standby_power_system_sObjectName                              :T_BA_StateText:='ESA';
  TxTPlant_Standby_power_system_sDescription                              :T_BA_StateText:='Ersatzstromanlage';
  TxTPlant_Photovoltaic_system_sObjectName                               :T_BA_StateText:='PVA';
  TxTPlant_Photovoltaic_system_sDescription                               :T_BA_StateText:='Fotovoltaikanlage';
  TxTPlant_Uninterruptible_power_supply_sObjectName                      :T_BA_StateText:='USV';
  TxTPlant_Uninterruptible_power_supply_sDescription                      :T_BA_StateText:='Unterbrechungsfreie Stromversorgung';
// 443 Niederspannungsschaltanlagen
  TxTPlant_General_power_supply_sObjectName                              :T_BA_StateText:='ASV';
  TxTPlant_General_power_supply_sDescription                              :T_BA_StateText:='Allgemeine Stromversorgung';
  TxTPlant_Safety_power_supply_sObjectName                               :T_BA_StateText:='SSV';
  TxTPlant_Safety_power_supply_sDescription                               :T_BA_StateText:='Sicherheitsstromversorgung';
  TxTPlant_Lighting_sObjectName                                          :T_BA_StateText:='BEL';
  TxTPlant_Lighting_sDescription                                          :T_BA_StateText:='Beleuchtungsanlage';
  TxTPlant_Emergency_lighting_sObjectName                                :T_BA_StateText:='SIB';
  TxTPlant_Emergency_lighting_sDescription                                :T_BA_StateText:='Sicherheitsbeleuchtung';
// 451 Telekommunikationsanlagen
  TxTPlant_Telecommunications_system_sObjectName                         :T_BA_StateText:='TEL';
  TxTPlant_Telecommunications_system_sDescription                         :T_BA_StateText:='Telekommunikationsanlage';
// 452 Such- und Signalanlagen
  TxTPlant_Call_signalling_system_sObjectName                            :T_BA_StateText:='LRA';
  TxTPlant_Call_signalling_system_sDescription                            :T_BA_StateText:='Lichtrufanlage';
  TxTPlant_Door_intercom_and_door_opener_system_sObjectName              :T_BA_StateText:='TÜA';
  TxTPlant_Door_intercom_and_door_opener_system_sDescription              :T_BA_StateText:='Türsprech- und -öffneranlage';
  TxTPlant_Paging_system_sObjectName                                     :T_BA_StateText:='PRA';
  TxTPlant_Paging_system_sDescription                                     :T_BA_StateText:='Personenrufanlage';
// 453 Zeitdienstanlagen
  TxTPlant_Clock_and_time_recording_system_sObjectName                   :T_BA_StateText:='ZEA';
  TxTPlant_Clock_and_time_recording_system_sDescription                   :T_BA_StateText:='Uhren- und Zeiterfassungsanlage';
// 454 Elektroakustische Anlagen
  TxTPlant_Electro_acoustic_sound_systems_sObjectName                    :T_BA_StateText:='ELA';
  TxTPlant_Electro_acoustic_sound_systems_sDescription                    :T_BA_StateText:='Elektroakustische Anl. , Beschallung';
  TxTPlant_Conference_and_interpreting_equipment_sObjectName             :T_BA_StateText:='KDA';
  TxTPlant_Conference_and_interpreting_equipment_sDescription             :T_BA_StateText:='Konferenz- und Dolmetscheranlage';
  TxTPlant_Intercom_system_sObjectName                                   :T_BA_StateText:='GSA';
  TxTPlant_Intercom_system_sDescription                                   :T_BA_StateText:='Gegensprechanlage';
  TxTPlant_Voice_alarm_system_sObjectName                                :T_BA_StateText:='SAA';
  TxTPlant_Voice_alarm_system_sDescription                                :T_BA_StateText:='Sprachalarmierungsanlage';
  TxTPlant_Intercommunication_systems_sObjectName                        :T_BA_StateText:='WSA';
  TxTPlant_Intercommunication_systems_sDescription                        :T_BA_StateText:='Wechselsprechanlagen';
// 455 Fernseh- und Antennenanlagen
  TxTPlant_Television_system_sObjectName                                 :T_BA_StateText:='TVA';
  TxTPlant_Television_system_sDescription                                 :T_BA_StateText:='Fernsehanlage';
  TxTPlant_Transmitting_and_receiving_antenna_system_sObjectName         :T_BA_StateText:='SEA';
  TxTPlant_Transmitting_and_receiving_antenna_system_sDescription         :T_BA_StateText:='Sende- und Empfangsantennenanlage';
  TxTPlant_BOS_radio_system_sObjectName                                  :T_BA_StateText:='BOS';
  TxTPlant_BOS_radio_system_sDescription                                  :T_BA_StateText:='BOS-Funkanlage';
// 456 Gefahrenmelde- und Alarmanlagen
  TxTPlant_Fire_detection_and_alarm_system_sObjectName                   :T_BA_StateText:='BMA';
  TxTPlant_Fire_detection_and_alarm_system_sDescription                   :T_BA_StateText:='Brandmeldeanlage';
  TxTPlant_Carbon_monoxide_warning_system_sObjectName                    :T_BA_StateText:='COW';
  TxTPlant_Carbon_monoxide_warning_system_sDescription                    :T_BA_StateText:='CO-Warnanlage';
  TxTPlant_Burglar_alarm_system_sObjectName                              :T_BA_StateText:='EMA';
  TxTPlant_Burglar_alarm_system_sDescription                              :T_BA_StateText:='Einbruchmeldeanlage';
  TxTPlant_Fire_control_panel_sObjectName                                :T_BA_StateText:='FWT';
  TxTPlant_Fire_control_panel_sDescription                                :T_BA_StateText:='Feuerwehrtableau';
  TxTPlant_Escape_route_protection_system_sObjectName                    :T_BA_StateText:='FWS';
  TxTPlant_Escape_route_protection_system_sDescription                    :T_BA_StateText:='Fluchtwegsicherungsanlage';
  TxTPlant_Hazard_detection_system_sObjectName                           :T_BA_StateText:='GMA';
  TxTPlant_Hazard_detection_system_sDescription                           :T_BA_StateText:='Gefahrenmeldeanlage';
  TxTPlant_Gas_warning_system_sObjectName                                :T_BA_StateText:='GWA';
  TxTPlant_Gas_warning_system_sDescription                                :T_BA_StateText:='Gaswarnanlage';
  TxTPlant_Smoke_aspiration_system_sObjectName                           :T_BA_StateText:='RAS';
  TxTPlant_Smoke_aspiration_system_sDescription                           :T_BA_StateText:='Rauchansaugsystem';
  TxTPlant_Room_observation_system_sObjectName                           :T_BA_StateText:='RBA';
  TxTPlant_Room_observation_system_sDescription                           :T_BA_StateText:='Raumbeobachtungsanlage';
  TxTPlant_Robbery_alarm_system_sObjectName                              :T_BA_StateText:='ÜFA';
  TxTPlant_Robbery_alarm_system_sDescription                              :T_BA_StateText:='Überfallmeldeanlage';
  TxTPlant_Guard_control_system_sObjectName                              :T_BA_StateText:='WKA';
  TxTPlant_Guard_control_system_sDescription                              :T_BA_StateText:='Wächterkontrollanlage';
  TxTPlant_Emergency_call_system_sObjectName                             :T_BA_StateText:='NOT';
  TxTPlant_Emergency_call_system_sDescription                             :T_BA_StateText:='Notrufanlage';
  TxTPlant_Access_control_system_sObjectName                             :T_BA_StateText:='ZKS';
  TxTPlant_Access_control_system_sDescription                             :T_BA_StateText:='Zugangskontrollsystem';
// 457 Übertragungsnetze
  TxTPlant_Networks_for_the_transmission_voice_text_etc_sObjectName      :T_BA_StateText:='LAN';
  TxTPlant_Networks_for_the_transmission_voice_text_etc_sDescription      :T_BA_StateText:='Netzw.  Daten, Sprache, Text etc';
// 459 Fernmelde- und informationstechnische Anlagen, Sonstiges
  TxTPlant_Remote_control_systems_sObjectName                            :T_BA_StateText:='FWA';
  TxTPlant_Remote_control_systems_sDescription                            :T_BA_StateText:='Fernwirkanlagen';
  TxTPlant_Parking_guidance_systems_sObjectName                          :T_BA_StateText:='PLS';
  TxTPlant_Parking_guidance_systems_sDescription                          :T_BA_StateText:='Parkleitsysteme';
// 460 Förderanlagen
  TxTPlant_File_transportation_systems_sObjectName                       :T_BA_StateText:='ATA';
  TxTPlant_File_transportation_systems_sDescription                       :T_BA_StateText:='Aktentransportanlagen';
  TxTPlant_Lift_sObjectName                                              :T_BA_StateText:='AUF';
  TxTPlant_Lift_sDescription                                              :T_BA_StateText:='Aufzug';
  TxTPlant_Inspection_systems_sObjectName                                :T_BA_StateText:='BFA';
  TxTPlant_Inspection_systems_sDescription                                :T_BA_StateText:='Befahranlagen';
  TxTPlant_Moving_walkways_sObjectName                                   :T_BA_StateText:='FST';
  TxTPlant_Moving_walkways_sDescription                                   :T_BA_StateText:='Fahrsteige';
  TxTPlant_Escalators_sObjectName                                        :T_BA_StateText:='FTR';
  TxTPlant_Escalators_sDescription                                        :T_BA_StateText:='Fahrtreppen';
  TxTPlant_External_lifts_sObjectName                                    :T_BA_StateText:='FSA';
  TxTPlant_External_lifts_sDescription                                    :T_BA_StateText:='Fassadenaufzüge';
  TxTPlant_Baggage_conveyor_system_sObjectName                           :T_BA_StateText:='GFA';
  TxTPlant_Baggage_conveyor_system_sDescription                           :T_BA_StateText:='Gepäckförderanlage';
  TxTPlant_Pneumatic_delivery_systems_sObjectName                        :T_BA_StateText:='RPA';
  TxTPlant_Pneumatic_delivery_systems_sDescription                        :T_BA_StateText:='Rohrpostanlagen';
  TxTPlant_Goods_transportation_facilities_sObjectName                   :T_BA_StateText:='WTA';
  TxTPlant_Goods_transportation_facilities_sDescription                   :T_BA_StateText:='Warentransportanlagen';
// 470 Nutzerspezifische Anlagen
// 471 Küchentechnische Anlagen
  TxTPlant_Small_refrigeration_unit_sObjectName                          :T_BA_StateText:='KLK';
  TxTPlant_Small_refrigeration_unit_sDescription                          :T_BA_StateText:='Kleinkälteanlage';
// 472 Wäscherei- und Reinigungsanlagen
  TxTPlant_Disinfection_unit_sObjectName                                 :T_BA_StateText:='DES';
  TxTPlant_Disinfection_unit_sDescription                                 :T_BA_StateText:='Desinfektionsanlage';
  TxTPlant_Cleaning_unit_sObjectName                                     :T_BA_StateText:='REA';
  TxTPlant_Cleaning_unit_sDescription                                     :T_BA_StateText:='Reinigungsanlage';
  TxTPlant_Sterilisation_systems_sObjectName                             :T_BA_StateText:='STR';
  TxTPlant_Sterilisation_systems_sDescription                             :T_BA_StateText:='Sterilisationseinrichtungen';
  TxTPlant_Water_treatment_system_sObjectName                            :T_BA_StateText:='WAA';
  TxTPlant_Water_treatment_system_sDescription                            :T_BA_StateText:='Wasseraufbereitungsanlage';
  TxTPlant_Laundry_system_sObjectName                                    :T_BA_StateText:='WÄA';
  TxTPlant_Laundry_system_sDescription                                    :T_BA_StateText:='Wäschereianlage';
// 473 Medienversorgungsanlagen
  TxTPlant_Compressed_air_supply_system_sObjectName                      :T_BA_StateText:='DRL';
  TxTPlant_Compressed_air_supply_system_sDescription                      :T_BA_StateText:='Druckluftversorgungsanlage';
  TxTPlant_Pressure_regulator_unit_sObjectName                           :T_BA_StateText:='DRA';
  TxTPlant_Pressure_regulator_unit_sDescription                           :T_BA_StateText:='Druckregelanlage';
  TxTPlant_Media_supply_system_sObjectName                               :T_BA_StateText:='MVA';
  TxTPlant_Media_supply_system_sDescription                               :T_BA_StateText:='Medienversorgungsanlage';
  TxTPlant_Medical_and_technical_gases_sObjectName                       :T_BA_StateText:='MTG';
  TxTPlant_Medical_and_technical_gases_sDescription                       :T_BA_StateText:='Medizinische und technische Gase';
  TxTPlant_Vacuum_unit_sObjectName                                       :T_BA_StateText:='VAK';
  TxTPlant_Vacuum_unit_sDescription                                       :T_BA_StateText:='Vakuumanlage';
// 474 Medizin- und labortechnische Anlagen
  TxTPlant_Medical_technical_plant_sObjectName                           :T_BA_StateText:='MED';
  TxTPlant_Medical_technical_plant_sDescription                           :T_BA_StateText:='Medizintechnische Anlagen';
  TxTPlant_Medical_gas_supply_sObjectName                                :T_BA_StateText:='MGV';
  TxTPlant_Medical_gas_supply_sDescription                                :T_BA_StateText:='Medizinische Gasversorgung';
  TxTPlant_Laboratory_equipment_sObjectName                              :T_BA_StateText:='LAB';
  TxTPlant_Laboratory_equipment_sDescription                              :T_BA_StateText:='Labortechnische Anlagen (allgemein)';
// 475 Feuerlöschanlagen
  TxTPlant_Fire_extinguisher_sObjectName                                 :T_BA_StateText:='FLA';
  TxTPlant_Fire_extinguisher_sDescription                                 :T_BA_StateText:='Feuerlöschanlage';
  TxTPlant_Gas_extinguishing_system_sObjectName                          :T_BA_StateText:='GLA';
  TxTPlant_Gas_extinguishing_system_sDescription                          :T_BA_StateText:='Gaslöschanlage';
  TxTPlant_Fire_extinguishing_system_sObjectName                         :T_BA_StateText:='LÖS';
  TxTPlant_Fire_extinguishing_system_sDescription                         :T_BA_StateText:='Löschanlage (allgemein)';
  TxTPlant_Mist_extinguishing_system_sObjectName                         :T_BA_StateText:='NLA';
  TxTPlant_Mist_extinguishing_system_sDescription                         :T_BA_StateText:='Nebellöschanlage';
  TxTPlant_NOX_system_sObjectName                                        :T_BA_StateText:='NOX';
  TxTPlant_NOX_system_sDescription                                        :T_BA_StateText:='NOX-Anlage';
  TxTPlant_Sprinkler_system_sObjectName                                  :T_BA_StateText:='SPR';
  TxTPlant_Sprinkler_system_sDescription                                  :T_BA_StateText:='Sprinkleranlage';
  TxTPlant_Wall_hydrant_system_sObjectName                               :T_BA_StateText:='WHA';
  TxTPlant_Wall_hydrant_system_sDescription                               :T_BA_StateText:='Wandhydrantenanlage';
// 478 Entsorgungsanlagen
  TxTPlant_Waste_disposal_system_sObjectName                             :T_BA_StateText:='AEA';
  TxTPlant_Waste_disposal_system_sDescription                             :T_BA_StateText:='Abfallentsorgungsanlage';
  TxTPlant_Media_disposal_system_sObjectName                             :T_BA_StateText:='MEA';
  TxTPlant_Media_disposal_system_sDescription                             :T_BA_StateText:='Medienentsorgungsanlage';
  TxTPlant_Vacuum_cleaning_systems_sObjectName                           :T_BA_StateText:='SSA';
  TxTPlant_Vacuum_cleaning_systems_sDescription                           :T_BA_StateText:='Staubsauganlagen';
// 480 Gebäudeautomation
  TxTPlant_Automation_control_equipment_sObjectName                      :T_BA_StateText:='ASP';
  TxTPlant_Automation_control_equipment_sDescription                      :T_BA_StateText:='Automationsschwerpunkt';
  TxTPlant_Weather_station_sObjectName                                   :T_BA_StateText:='WET';
  TxTPlant_Weather_station_sDescription                                   :T_BA_StateText:='Wetterstation';
  TxTPlant_Management_and_operating_equipment_sObjectName                :T_BA_StateText:='MBE';
  TxTPlant_Management_and_operating_equipment_sDescription                :T_BA_StateText:='Management- und Bedieneinrichtungen';
  TxTPlant_Room_automation_sObjectName                                   :T_BA_StateText:='RAU';
  TxTPlant_Room_automation_sDescription                                   :T_BA_StateText:='Raumautomation';
  TxTPlant_Room_automation_system_distributor_sObjectName                :T_BA_StateText:='RAV';
  TxTPlant_Room_automation_system_distributor_sDescription                :T_BA_StateText:='Raumautomation-Systemverteiler';
  TxTPlant_Control_cabinet_sObjectName                                   :T_BA_StateText:='SSK';
  TxTPlant_Control_cabinet_sDescription                                   :T_BA_StateText:='Schaltschrank';
  TxTPlant_Settings_sObjectName                                          :T_BA_StateText:='ALP';
  TxTPlant_Settings_sDescription                                          :T_BA_StateText:='Anlagenparameter';
  TxTPlant_EventGroups_sObjectName                                       :T_BA_StateText:='ERG';
  TxTPlant_EventGroups_sDescription                                       :T_BA_StateText:='Meldeklassen';
  TxTPlant_Global_Building_Data_sObjectName                              :T_BA_StateText:='GGL';
  TxTPlant_Global_Building_Data_sDescription                              :T_BA_StateText:='globale Gebäudedaten';
// 540 Technische Anlagen in Außenanlagen
  TxTPlant_Rainwater_retention_basin_sObjectName                         :T_BA_StateText:='RRB';
  TxTPlant_Rainwater_retention_basin_sDescription                         :T_BA_StateText:='Regenrückhaltebecken';
  TxTPlant_Cistern_system_sObjectName                                    :T_BA_StateText:='ZTA';
  TxTPlant_Cistern_system_sDescription                                    :T_BA_StateText:='Zisternenanlage';
END_VAR

// ---- Templates/GVLs/Language/German/TxtTrade_DE.TcGVL
{region '#Template'}
	{attribute 'Version' := '5.0.0.0'}
	{attribute 'Tags' := '"LCID": "1031", "Text": "GVL, DPAD, Trades, ObjectName, Description"'}
	{attribute 'Tags' := '"LCID": "1033", "Text": "GVL, DPAD, Trades, ObjectName, Description"'}
	{attribute 'Description' := '"LCID": "1031", "Text": "Textliste Gewerke"'}
	{attribute 'Description' := '"LCID": "1033", "Text": "Text list trades"'}
{endregion}

{attribute 'global_init_slot' := '40510'}
VAR_GLOBAL
  TxtTrade_Doors_gates_windows_sun_protection_sObjectName                :T_BA_StateText:='TTF';
  TxtTrade_Doors_gates_windows_sun_protection_sDescription                :T_BA_StateText:='Türen, Tore, Fenster, Sonnenschutz';
  TxtTrade_Sewage_water_and_gas_plants_sObjectName                       :T_BA_StateText:='GWA';
  TxtTrade_Sewage_water_and_gas_plants_sDescription                       :T_BA_StateText:='Abwasser-, Wasser-, Gasanlagen';
  TxtTrade_Heat_supply_systems_sObjectName                               :T_BA_StateText:='HZG';
  TxtTrade_Heat_supply_systems_sDescription                               :T_BA_StateText:='Wärmeversorgungsanlagen';
  TxtTrade_Air_conditioning_sObjectName                                  :T_BA_StateText:='LTA';
  TxtTrade_Air_conditioning_sDescription                                  :T_BA_StateText:='Lufttechnische Anlagen';
  TxtTrade_Refrigeration_systems_sObjectName                             :T_BA_StateText:='KAE';
  TxtTrade_Refrigeration_systems_sDescription                             :T_BA_StateText:='Kälteanlagen';
  TxtTrade_High_voltage_systems_sObjectName                              :T_BA_StateText:='ELT';
  TxtTrade_High_voltage_systems_sDescription                              :T_BA_StateText:='Starkstromanlagen';
  TxtTrade_Telecommunication_and_information_technology_sObjectName      :T_BA_StateText:='FIA';
  TxtTrade_Telecommunication_and_information_technology_sDescription      :T_BA_StateText:='Fernm.- und informationstech. Anlagen';
  TxtTrade_Hazard_detection_and_alarm_systems_sObjectName                :T_BA_StateText:='GMA';
  TxtTrade_Hazard_detection_and_alarm_systems_sDescription                :T_BA_StateText:='Gefahrenmelde- und Alarmanlagen';
  TxtTrade_Conveyors_sObjectName                                         :T_BA_StateText:='FTA';
  TxtTrade_Conveyors_sDescription                                         :T_BA_StateText:='Förderanlagen';
  TxtTrade_Kitchen_technology_systems_sObjectName                        :T_BA_StateText:='KTA';
  TxtTrade_Kitchen_technology_systems_sDescription                        :T_BA_StateText:='Küchentechnische Anlagen';
  TxtTrade_Laundry_and_cleaning_systems_sObjectName                      :T_BA_StateText:='WAR';
  TxtTrade_Laundry_and_cleaning_systems_sDescription                      :T_BA_StateText:='Wäscherei- und Reinigungsanlagen';
  TxtTrade_Media_supply_systems_sObjectName                              :T_BA_StateText:='MVA';
  TxtTrade_Media_supply_systems_sDescription                              :T_BA_StateText:='Medienversorgungsanlagen';
  TxtTrade_Medical_and_laboratory_equipment_sObjectName                  :T_BA_StateText:='MED';
  TxtTrade_Medical_and_laboratory_equipment_sDescription                  :T_BA_StateText:='Medizin- und labortechnische Anlagen';
  TxtTrade_Fire_extinguishing_systems_sObjectName                        :T_BA_StateText:='FLA';
  TxtTrade_Fire_extinguishing_systems_sDescription                        :T_BA_StateText:='Feuerlöschanlagen';
  TxtTrade_Bathing_facilities_sObjectName                                :T_BA_StateText:='BTA';
  TxtTrade_Bathing_facilities_sDescription                                :T_BA_StateText:='Badetechnische Anlagen';
  TxtTrade_Process_heating_cooling_and_air_systems_sObjectName           :T_BA_StateText:='PRO';
  TxtTrade_Process_heating_cooling_and_air_systems_sDescription           :T_BA_StateText:='Prozesswärme-, -kälte- und -luftanlagen';
  TxtTrade_Waste_disposal_facilities_sObjectName                         :T_BA_StateText:='ENT';
  TxtTrade_Waste_disposal_facilities_sDescription                         :T_BA_StateText:='Entsorgungsanlagen';
  TxtTrade_Building_automation_and_control_systems_general_sObjectName   :T_BA_StateText:='GAS';
  TxtTrade_Building_automation_and_control_systems_general_sDescription   :T_BA_StateText:='Gebäudeautomation allgemein';
  TxtTrade_Automation_focal_point_information_focal_point_sObjectName    :T_BA_StateText:='ASP';
  TxtTrade_Automation_focal_point_information_focal_point_sDescription    :T_BA_StateText:='Automationsschwerpunkt';
  TxtTrade_Room_automation_sObjectName                                   :T_BA_StateText:='RAU';
  TxtTrade_Room_automation_sDescription                                   :T_BA_StateText:='Raumautomation';
  TxtTrade_Outdoor_devices_sObjectName                                   :T_BA_StateText:='AUG';
  TxtTrade_Outdoor_devices_sDescription                                   :T_BA_StateText:='Außengeräte';
END_VAR

// ---- Templates/GVLs/LblComp.TcGVL
{region '#Template'}
	{attribute 'Version' := '5.1.0.0'}
	{attribute 'Tags' := '"LCID": "1031", "Text": "GVL, Kompositionen von Labels für Sonderfunktionen"'}
	{attribute 'Tags' := '"LCID": "1033", "Text": "GVL, LabelComposition for Secial Functions"'}
	{attribute 'Description' := '"LCID": "1031", "Text": "Label Kompositionen"'}
	{attribute 'Description' := '"LCID": "1033", "Text": "Label composition"'}
{endregion}

{attribute 'global_init_slot' := '40520'}
VAR_GLOBAL
	LblComp_Project								:FB_BA_Label2x:=(iAggregate:=LblAgg_AutomationStationEquipment,	iFunction:=LblCTL_BACnetDevice);
	
	//     Composition of 2 Labels
	//     479 User-specific system, weather station 
	LblComp_Wth_RainSensor						:FB_BA_Label2x:=(iAggregate:=LblAgg_RainSensor,			iFunction:=LblFun_OperationalMessage);
	LblComp_Wth_WeatherStation					:FB_BA_Label2x:=(iAggregate:=LblAgg_WeatherStation,		iFunction:=LblFun_Fault);
												
	LblComp_Wth_TemperatureOutside				:FB_BA_Label2x:=(iAggregate:=LblAgg_TemperatureOutside,	iFunction:=LblFun_MeasuredValue);
	LblComp_Wth_TemperatureDewPoint				:FB_BA_Label2x:=(iAggregate:=LblAgg_TemperatureDewPoint,iFunction:=LblFun_MeasuredValue);
	LblComp_Wth_PressureAbsolute				:FB_BA_Label2x:=(iAggregate:=LblAgg_PressureAbsolute,	iFunction:=LblFun_MeasuredValue);
	LblComp_Wth_PressureRelative				:FB_BA_Label2x:=(iAggregate:=LblAgg_PressureRelative,	iFunction:=LblFun_MeasuredValue);
	LblComp_Wth_AbsoluteHumidityOutsideAir		:FB_BA_Label2x:=(iAggregate:=LblAgg_AbsoluteHumidityOutsideAir,iFunction:=LblFun_MeasuredValue);
	LblComp_Wth_RelativeHumidityOutsideAir		:FB_BA_Label2x:=(iAggregate:=LblAgg_RelativeHumidityOutsideAir,iFunction:=LblFun_MeasuredValue);
	LblComp_Wth_Brightness						:FB_BA_Label2x:=(iAggregate:=LblAgg_Brightness,			iFunction:=LblFun_MeasuredValue);
	LblComp_Wth_Dawn							:FB_BA_Label2x:=(iAggregate:=LblAgg_Dawn,				iFunction:=LblFun_MeasuredValue);
	LblComp_Wth_SolarRadiation					:FB_BA_Label2x:=(iAggregate:=LblAgg_SolarRadiation,		iFunction:=LblFun_MeasuredValue);
	LblComp_Wth_WindDirection					:FB_BA_Label2x:=(iAggregate:=LblAgg_WindDirection,		iFunction:=LblFun_MeasuredValue);
	LblComp_Wth_WindSpeed						:FB_BA_Label2x:=(iAggregate:=LblAgg_WindSpeed,			iFunction:=LblFun_MeasuredValue);
	LblComp_Wth_GeoLatitude						:FB_BA_Label2x:=(iAggregate:=LblAgg_GeoLatitude,		iFunction:=LblFun_MeasuredValue);
	LblComp_Wth_GeoLongitude					:FB_BA_Label2x:=(iAggregate:=LblAgg_GeoLongitude,		iFunction:=LblFun_MeasuredValue);
	LblComp_Wth_SunAzimuth						:FB_BA_Label2x:=(iAggregate:=LblAgg_SunAzimuth,			iFunction:=LblFun_MeasuredValue);
	LblComp_Wth_SunElevation					:FB_BA_Label2x:=(iAggregate:=LblAgg_SunElevation,		iFunction:=LblFun_MeasuredValue);
	
	LblComp_Wth_WeatherStationReset       		:FB_BA_Label2x:=(iAggregate:=LblAgg_WeatherStationReset,iFunction:=LblFun_SwitchingCommand);
	LblComp_Wth_WeatherStationCommReset   		:FB_BA_Label2x:=(iAggregate:=LblAgg_WeatherStationCommReset,iFunction:=LblFun_SwitchingCommand);
	LblComp_Wth_WeatherStationComm        		:FB_BA_Label2x:=(iAggregate:=LblAgg_WeatherStationComm,	iFunction:=LblFun_Fault);  


	// Temperature // Temperatur
	LblComp_TempExtA_MV        			   		:FB_BA_Label2x:=(iAggregate:=LblAgg_TemperatureExtractAir,		iFunction:=LblFun_MeasuredValue);  
	LblComp_TempExhA_MV        			   		:FB_BA_Label2x:=(iAggregate:=LblAgg_TemperatureExhaustAir,		iFunction:=LblFun_MeasuredValue);  
	LblComp_TempOuA_MV        			   		:FB_BA_Label2x:=(iAggregate:=LblAgg_TemperatureOutside,			iFunction:=LblFun_MeasuredValue);  
	LblComp_TempRmA_MV        			   		:FB_BA_Label2x:=(iAggregate:=LblAgg_TemperatureRoomAir,			iFunction:=LblFun_MeasuredValue);  
	LblComp_TempSuA_MV        			   		:FB_BA_Label2x:=(iAggregate:=LblAgg_TemperatureSupplyAir,		iFunction:=LblFun_MeasuredValue);  
	
	// Relative humidity // Relative Feuchte
	LblComp_RelHumExtA_MV        			   	:FB_BA_Label2x:=(iAggregate:=LblAgg_RelativeHumidityExtractAir,		iFunction:=LblFun_MeasuredValue);  
	LblComp_RelHumExhA_MV        			   	:FB_BA_Label2x:=(iAggregate:=LblAgg_RelativeHumidityExhaustAir,		iFunction:=LblFun_MeasuredValue);  
	LblComp_RelHumOuA_MV        			   	:FB_BA_Label2x:=(iAggregate:=LblAgg_RelativeHumidityOutsideAir,		iFunction:=LblFun_MeasuredValue);  
	LblComp_RelHumRmA_MV        			   	:FB_BA_Label2x:=(iAggregate:=LblAgg_RelativeHumidityRoomHumidity,	iFunction:=LblFun_MeasuredValue);  
	LblComp_RelHumSuA_MV        			   	:FB_BA_Label2x:=(iAggregate:=LblAgg_RelativeHumiditySupplyAir,		iFunction:=LblFun_MeasuredValue);  
	
	// Absolute humidity // Absolute Feuchte
	LblComp_AbsHumExtA_MVC       			   	:FB_BA_Label2x:=(iAggregate:=LblAgg_AbsoluteHumidityExtractAir,	iFunction:=LblFun_MeasuredValueCalculated);  
	LblComp_AbsHumExhA_MVC       			   	:FB_BA_Label2x:=(iAggregate:=LblAgg_AbsoluteHumidityExhaustAir,	iFunction:=LblFun_MeasuredValueCalculated);  
	LblComp_AbsHumOuA_MVC        			   	:FB_BA_Label2x:=(iAggregate:=LblAgg_AbsoluteHumidityOutsideAir,	iFunction:=LblFun_MeasuredValueCalculated);  
	LblComp_AbsHumRmA_MVC        			   	:FB_BA_Label2x:=(iAggregate:=LblAgg_AbsoluteHumidityRoomAir,	iFunction:=LblFun_MeasuredValueCalculated);  
	LblComp_AbsHumSuA_MVC        			   	:FB_BA_Label2x:=(iAggregate:=LblAgg_AbsoluteHumiditySupplyAir,	iFunction:=LblFun_MeasuredValueCalculated);  
	
	// Dew point temperature // Taupunkttemperatur
	LblComp_DewPntExtA_MVC       			   	:FB_BA_Label2x:=(iAggregate:=LblAgg_TemperatureDewPointExtractAir,	iFunction:=LblFun_MeasuredValueCalculated);  
	LblComp_DewPntExhA_MVC       			   	:FB_BA_Label2x:=(iAggregate:=LblAgg_TemperatureDewPointExhaustAir,	iFunction:=LblFun_MeasuredValueCalculated);  
	LblComp_DewPntOuA_MVC        			   	:FB_BA_Label2x:=(iAggregate:=LblAgg_TemperatureDewPointOutsideAir,	iFunction:=LblFun_MeasuredValueCalculated);  
	LblComp_DewPntRmA_MVC        			   	:FB_BA_Label2x:=(iAggregate:=LblAgg_TemperatureDewPointRoomAir,	iFunction:=LblFun_MeasuredValueCalculated);  
	LblComp_DewPntSuA_MVC        			   	:FB_BA_Label2x:=(iAggregate:=LblAgg_TemperatureDewPointSupplyAir,	iFunction:=LblFun_MeasuredValueCalculated);  
	
	// Enthalpy // Enthalpie
	LblComp_EnthalpyExtA_MVC       			   	:FB_BA_Label2x:=(iAggregate:=LblAgg_EnthalpyExtractAir,	iFunction:=LblFun_MeasuredValueCalculated);  
	LblComp_EnthalpyExhA_MVC       			   	:FB_BA_Label2x:=(iAggregate:=LblAgg_EnthalpyExhaustAir,	iFunction:=LblFun_MeasuredValueCalculated);  
	LblComp_EnthalpyOuA_MVC        			   	:FB_BA_Label2x:=(iAggregate:=LblAgg_EnthalpyOutsideAir,	iFunction:=LblFun_MeasuredValueCalculated);  
	LblComp_EnthalpyRmA_MVC        			   	:FB_BA_Label2x:=(iAggregate:=LblAgg_EnthalpyRoomAir,	iFunction:=LblFun_MeasuredValueCalculated);  
	LblComp_EnthalpySuA_MVC        			   	:FB_BA_Label2x:=(iAggregate:=LblAgg_EnthalpySupplyAir,	iFunction:=LblFun_MeasuredValueCalculated);  
	
	// Wet bulp temperature // Feuchtkugeltemperatur
	LblComp_TempWetBulpExtA_MVC       	   		:FB_BA_Label2x:=(iAggregate:=LblAgg_TemperatureWetBulpExtractAir,	iFunction:=LblFun_MeasuredValueCalculated);  
	LblComp_TempWetBulpExhA_MVC       	   		:FB_BA_Label2x:=(iAggregate:=LblAgg_TemperatureWetBulpExhaustAir,	iFunction:=LblFun_MeasuredValueCalculated);  
	LblComp_TempWetBulpOuA_MVC        	   		:FB_BA_Label2x:=(iAggregate:=LblAgg_TemperatureWetBulpOutsideAir,	iFunction:=LblFun_MeasuredValueCalculated);  
	LblComp_TempWetBulpRmA_MVC        	   		:FB_BA_Label2x:=(iAggregate:=LblAgg_TemperatureWetBulpRoomAir,		iFunction:=LblFun_MeasuredValueCalculated);  
	LblComp_TempWetBulpSuA_MVC        	   		:FB_BA_Label2x:=(iAggregate:=LblAgg_TemperatureWetBulpSupplyAir,	iFunction:=LblFun_MeasuredValueCalculated);  
END_VAR

// ---- Templates/GVLs/Site/Site.TcGVL
{region '#Template'}
	{attribute 'Version' := '5.1.1.0'}
	{attribute 'Tags' := '"LCID": "1031", "Text": "GVL, Publisher, Subscriber"'}
	{attribute 'Tags' := '"LCID": "1033", "Text": "GVL, Publisher, Subscriber"'}
	{attribute 'Using' := '"Type": "Template", "URI": "ST_BA_GeneralSettings"'}
	{attribute 'Using' := '"Type": "Template", "URI": "E_BA_EnergyLvlEx"'}
	{attribute 'Using' := '"Type": "Template", "URI": "E_BA_BuildingMode"'}
	{attribute 'Using' := '"Type": "Template", "URI": "ST_BA_BuildingSunBlind"'}
	{attribute 'Using' := '"Type": "Template", "URI": "ST_BA_BuildingAlarms"'}
	{attribute 'Using' := '"Type": "Template", "URI": "ST_BA_WeatherStation"'}
	{attribute 'Using' := '"Type": "Template", "URI": "ST_BA_Facade"'}		 
	{attribute 'Description' := '"LCID": "1031", "Text": "Ams NetId, Subject"'}
	{attribute 'Description' := '"LCID": "1033", "Text": "Ams NetId, Subject"'}
{endregion}

{attribute 'qualified_only'}
VAR_GLOBAL	
	Self_NetId						: T_BA_MedString	:= '127.0.0.1.1.1';
	ACE01_NetId						: T_BA_MedString	:= Self_NetId;
	ACE02_NetId						: T_BA_MedString	:= Self_NetId;
	ACE03_NetId						: T_BA_MedString	:= Self_NetId;
	ACE04_NetId						: T_BA_MedString	:= Self_NetId;
	ACE05_NetId						: T_BA_MedString	:= Self_NetId;
	                            	
	GeneralSettings_Subject			: T_BA_MedString	:= 'GeneralSettings';	
	GeneralSettings_NetId			: T_BA_MedString	:= ACE01_NetId;	
		                        	
	WeatherStation_Subject			: T_BA_MedString	:= 'WeatherStation';
	WeatherStation_NetId			: T_BA_MedString	:= ACE01_NetId;
                                	
	FacadeNorth_Subject				: T_BA_MedString	:= 'arrFacadeData[1]';
	FacadeNorth_NetId				: T_BA_MedString	:= ACE01_NetId;
	FacadeEast_Subject				: T_BA_MedString	:= 'arrFacadeData[2]';
	FacadeEast_NetId				: T_BA_MedString	:= ACE01_NetId;
	FacadeSouth_Subject				: T_BA_MedString	:= 'arrFacadeData[3]';
	FacadeSouth_NetId				: T_BA_MedString	:= ACE01_NetId;
	FacadeWest_Subject				: T_BA_MedString	:= 'arrFacadeData[4]';
	FacadeWest_NetId				: T_BA_MedString	:= ACE01_NetId;
                                	
	Building_NetId					: T_BA_MedString	:= ACE01_NetId;
	BuildingAlarms_Subject			: T_BA_MedString	:= 'BuildingAlarms';
	BuildingMode_Subject			: T_BA_MedString	:= 'BuildingMode';
	BuildingEnergyLevel_Subject		: T_BA_MedString	:= 'BuildingEnergyLevel';
	BuildingSpRmT_Subject			: T_BA_MedString	:= 'BuildingSpRmT';
	BuildingSunBlind_Subject		: T_BA_MedString	:= 'BuildingSunBlind';
	BuildingLighting_Subject		: T_BA_MedString	:= 'BuildingLighting';
		
	
	stGeneralSettings				: ST_BA_GeneralSettings;	// provided by FB_BA_WeatherData	
	bGeneralSettings_Error			: BOOL;	
	stWeatherStation				: ST_BA_WeatherStation;		// provided by FB_BA_WeatherStation_xxx
	bWeatherStation_Error			: BOOL;
	stBuildingAlarms				: ST_BA_BuildingAlarms;		// provided by FB_BA_BurglarAlarmSystem and FB_BA_FireAlarmSystem
	bBuildingAlarms_Error			: BOOL;
	eBuildingMode					: E_BA_BuildingMode;		// provided by FB_BA_BuildingMode
	bBuildingMode_Error				: BOOL;
	eBuildingEnergyLevel			: E_BA_EnergyLvlEx;			// provided by FB_BA_BuildingEnergyLevel
	bBuildingEnergyLevel_Error		: BOOL;
	stBuildingSpRmT					: ST_BA_SpRmT;				// provided by FB_BA_BuildingSpRmT
	bBuildingSpRmT_Error			: BOOL;
	stBuildingSunBlind				: ST_BA_BuildingSunBlind;	// provided by FB_BA_BuildingSunprotection
	bBuildingSunBlind_Error			: BOOL;
	stBuildingLighting				: ST_BA_BuildingLighting;	// provided by FB_BA_BuildingLighting
	bBuildingLighting_Error			: BOOL;
	eHeatCoolMedium					: E_BA_Medium;				// actual medium running in case of a two-pipe-system
	bHeatCoolMedium_Error			: BOOL;	
	
	arrFacade 						: ARRAY  [1..BA2_Param.nMaxNumberOfFacades] OF ST_BA_Facade; 	//  provided by Array [1..BA2_Param.nMaxNumberOffFacades Of FB_BA_Facade] 
	arrFacade_Error					: ARRAY  [1..BA2_Param.nMaxNumberOfFacades] OF BOOL;
	
	arrAreaLighting					: ARRAY  [1..BA2_Param.nMaxNumberOfAreas]	OF ST_BA_Lighting;	//  provided by Array [1..BA2_Param.nMaxNumberOffFacades Of FB_BA_Lighting] 
END_VAR

// ---- Templates/GVLs/SysTime.TcGVL
{region '#Template'}
	{attribute 'Version' := '5.0.0.0'}
	{attribute 'Tags' := '"LCID": "1031", "Text": "GVL, Systemzeiten"'}
	{attribute 'Tags' := '"LCID": "1033", "Text": "GVL, System times"'}
	{attribute 'Description' := '"LCID": "1031", "Text": "Systemzeiten"'}
	{attribute 'Description' := '"LCID": "1033", "Text": "System times"'}
{endregion}

{attribute 'qualified_only'}
VAR_GLOBAL
	stSystemTime			: TIMESTRUCT;
	stSystemTimeUTC			: TIMESTRUCT;
	dtSystemTime			: DT;
	dtSystemTimeUTC			: DT;
END_VAR

// ---- POUs/DALICommunication.TcPOU
PROGRAM DALICommunication
VAR

	stKL6821InData			AT %I*	: Tc3_DALI.ST_KL6821InData;       
	stKL6821OutData			AT %Q*	: Tc3_DALI.ST_KL6821OutData;
	
	fbKL6821Communication			: Tc3_DALI.FB_KL6821Communication;
	
	bError							: BOOL;
	bResetMaximumDemandCounter		: BOOL;
	bResetOverflowCounter			: BOOL;
	nOptions						: DWORD;
	bBusy							: BOOL;
	nBufferDemandMeter				: BYTE;
	nBufferMaximumDemandMeter		: BYTE;
	nBufferOverflowCounter			: UINT;
	bResetInactiveProcessImage		: BOOL;
	bInitialise						: BOOL;
	nErrorId						: DWORD;
	
	bDigitalInput1Active			: BOOL;
	bDigitalInput2Active			: BOOL;
	bProcessImageInactive			: BOOL;
	bCollisionError					: BOOL;
	bPowerSupplyError				: BOOL;
	bShortCircuit					: BOOL;
	bInitialising					: BOOL;
	nTerminalDescription			: WORD;
	nFirmwareVersion				: WORD;
	
END_VAR


						
fbKL6821Communication(	bError							=> bError, 
						bResetMaximumDemandCounter		:= bResetMaximumDemandCounter, 
						bResetOverflowCounter			:= bResetOverflowCounter, 
						nOptions						:= nOptions, 
						bBusy							=> bBusy, 
						nBufferDemandMeter				=> nBufferDemandMeter, 
						nBufferMaximumDemandMeter		=> nBufferMaximumDemandMeter, 
						nBufferOverflowCounter			=> nBufferOverflowCounter, 
						bResetInactiveProcessImage		:= bResetInactiveProcessImage, 
						bInitialise						:= bInitialise, 
						bDigitalInput1Active			=> bDigitalInput1Active, 
						bDigitalInput2Active			=> bDigitalInput2Active, 
						bProcessImageInactive			=> bProcessImageInactive, 
						bCollisionError					=> bCollisionError, 
						bPowerSupplyError				=> bPowerSupplyError, 
						bShortCircuit					=> bShortCircuit, 
						bInitialising					=> bInitialising, 
						nTerminalDescription			=> nTerminalDescription, 
						nFirmwareVersion				=> nFirmwareVersion, 
						stInData						:= stKL6821InData, 
						stOutData						:= stKL6821OutData);

END_PROGRAM

// ---- POUs/MAIN.TcPOU
PROGRAM MAIN
VAR
DPAD		: FB_BA_CarelessDPAD := (
					aIdentifier := [
	(* Level 1 *)		(	eNodeType:=E_BA_NodeType.eBuilding,			sSeparator_ObjectName := '-', 	sSeparator_Description := ' - ',	nIndexDigits := 0),
	(* Level 2 *)		(	eNodeType:=E_BA_NodeType.eFloor,			sSeparator_ObjectName := '-', 	sSeparator_Description := ' - ',	nIndexDigits := 0),
	(* Level 3 *)		(	eNodeType:=E_BA_NodeType.eTrade,			sSeparator_ObjectName := '-', 	sSeparator_Description := ' - ',	nIndexDigits := 0),
	(* Level 4 *)		(	eNodeType:=E_BA_NodeType.ePlant,			sSeparator_ObjectName := '-', 	sSeparator_Description := ' - ',	nIndexDigits := 2),
	(* Level 5 *)		(	eNodeType:=E_BA_NodeType.eAggregate,		sSeparator_ObjectName := '-', 	sSeparator_Description := ' - ',	nIndexDigits := 2),
	(* Level 6 *)		(	eNodeType:=E_BA_NodeType.eFunction,			sSeparator_ObjectName := '-', 	sSeparator_Description := ' - ',	nIndexDigits := 2)
					]
				);
//	Level 1 Gebäude 	
//	Level 1 Building 	
		B			: FB_BA_View := (
						sObjectName		:= 'B',	
						sDescription	:= 'Building B'				
					);
// Level 2 Gebäudeteil
// Level 2 Part of building						
			PB1			: FB_BA_View := (
							iParent 		:= B,
							sObjectName		:= '{PB1}',		
							sDescription	:= '{Part of building 1}'			
						);   
// Level 3 Gewerk Automationsschwerpunkt
// Level 3 Trade AutomationFocalPoint                                                                                       	
				ACE			: FB_BA_AutomationControl := (
								iParent 		:= PB1,
								sObjectName		:= '{ACE}',
								sDescription	:= '{Automation Control}'								
							);
// Level 3 Gewerk Gebäudeautomation Allgemein	- SERVER
// Level 3 Trade building automation general	- SERVER                                                                       	
				BAG			: FB_BA_BuildingAutomationServer := (
								iParent 		:= PB1,
								sObjectName		:= '{BAG}',
								sDescription	:= '{Building Automation}'
							);    	
// Level 3 Gewerk Wärmeversorgungsanlagen  
// Level 3 Trade Heat supply systems, heat distribution  --> 	HD = heat distribution, HG = heat generation
				HTG			: FB_BA_Heating := (
								iParent 		:= PB1,
								sObjectName		:= '{HTG}',
								sDescription	:= '{Heating}'			
							);     	    
// Level 3 Gewerk Luftechnische Anlagen      
// Level 3 Trade ventilation system        
				ACS			: FB_BA_AirConditioning := (
								iParent 		:= PB1,
								sObjectName		:= '{ACS}',
								sDescription	:= '{Air Conditioning}'					
							);  			     
// Level 3 Gewerk Raumautomation	- SERVER
// Level 3 Trade room automation	- SERVER
				ROM			: FB_BA_RoomAutomationServer := (
								iParent			:= PB1,
								sObjectName		:= '{ROM}',
								sDescription	:= '{Room automation}'
							);
// Level 3 Gewerk Gefahrenmelde- und Alarmanlagen   
// Level 3 Trade Hazard Detection and Alarm Systems  				
				HDAS		: FB_BA_HazardDetectionAlarmSystems:= (
								iParent 		:= PB1,
								sObjectName		:= '{GMA}',
								sDescription	:= '{Hazard detection and alarm systems}'
							);
// Level 3 Gewerk Türen, Tore, Fenster, Sonnenschutz	- SERVER
// Level 3 Trade Doors, gates, windwos, sun protection	- SERVER
				DGWSP		: FB_BA_DGWSPServer := (
								iParent 		:= PB1,
								sObjectName		:= '{TTF}',
								sDescription	:= '{Doors - gates - windows - sun-protection}'
							);								
// SystemTime Settings								
	BACnetTime_TO_SysTime		: FB_BA_BACnetTime_TO_SysTime;	
	ExternalSysTime				: FB_BA_ExternalSysTime;
END_VAR

//	Level 1 Gebäude 	Building		
	B();
// Level 2 Gebäudeteil		Part of building
		PB1();
// Level 3 Gewerk Automation							Trade Automation			
			ACE(); 							
// Level 3 Gewerk Gebäudeautomation Allgemein			Trade BuildingAutomationGeneral			
			BAG(); 								
// Level 3 Gewerk Wärmeversorgungsanlagen				Trade Heat supply systems	
			HTG(); 	
// Level 3 Gewerk Lufttechnische Anlagen				Trade ventilation system	
			ACS(); 								
// Level 3 Gewerk Raumautomation						Trade room automation 
			ROM(); 		
// Level 3 Gewerk Gefahrenmelde- und Alarmanlagen		Trade Hazard detection and alarm systems
			HDAS();	
// Level 3 Gewerk Türen, Tore, Fenster, Sonnenschutz	Trade Doors, gates, windows, sun protection			
			DGWSP();	

//	BACnetTime_TO_SysTime();	
	ExternalSysTime();

END_PROGRAM

// ---- Templates/POUs/Trade/BuildingAutomation/FB_BA_BuildingAutomationServer.TcPOU
{region '#Template'}                                                                                                                                                                                                                                                {region '#Template'}
	{attribute 'Version' := '5.0.0.0'}
	{attribute 'Tags' := '"LCID": "1031", "Text": "Gewerk, Gebäudeautomation"'}
	{attribute 'Tags' := '"LCID": "1033", "Text": "Trade, Building automation"'}
	{attribute 'Using' := '"Type": "Template", "URI": "Site"'}
	{attribute 'Description' := '"LCID": "1031", "Text": "Aufruf der Anlagen des Gewerks Gebäudeautomation"'}
	{attribute 'Description' := '"LCID": "1033", "Text": "Calling the plants of the trade building automation"'}
{endregion}	 
	 
FUNCTION_BLOCK FB_BA_BuildingAutomationServer EXTENDS FB_BA_View
VAR_INPUT CONSTANT
	AdsComServerBasic		: FB_BA_AdsComServer_Basic;	
	Weatherstation01		: FB_BA_WeatherStation_Thies;	
	WeatherData 			: FB_BA_WeatherData;	
END_VAR

SUPER^(); // FB_BA_View
AdsComServerBasic(); // FB_BA_AdsComServer_Basic
Weatherstation01(); // FB_BA_WeatherStation_Thies
WeatherData(); // FB_BA_WeatherData

METHOD FB_init : BOOL
VAR_INPUT
	bInitRetains : BOOL; // if TRUE, the retain variables are initialized (warm start / cold start)
	bInCopyCode : BOOL;  // if TRUE, the instance afterwards gets moved into the copy code (online change)
END_VAR
Weatherstation01.iParent		:= THIS^;
Weatherstation01.iLabel			:= LblPlt_Weather_station;
Weatherstation01.sObjectName	:= '{Idx=01}';
Weatherstation01.sDescription	:= '{Idx=01}';
Weatherstation01.eDPADMode		:= E_BA_DPADMode.eInclude;

WeatherData.iParent			    := THIS^;
WeatherData.iLabel			    := LblPlt_Weather_data;
WeatherData.sObjectName		    := '{Idx=01}';
WeatherData.eDPADMode		    := E_BA_DPADMode.eInclude;
END_METHOD

END_FUNCTION_BLOCK

// ---- Templates/POUs/Trade/BuildingAutomation/Weather_Data/FB_BA_WeatherData.TcPOU
{region '#Template'}
	{attribute 'Version' := '5.0.0.0'}
	{attribute 'Tags' := '"LCID": "1031", "Text": "Gebäudeautomation, Wetterdaten"'}
	{attribute 'Tags' := '"LCID": "1033", "Text": "Building automation, Weather data"'}
	{attribute 'Using' := '"Type": "Template", "URI": "BA2_Param"'}
	{attribute 'Using' := '"Type": "Template", "URI": "Site"'}		  
	{attribute 'Using' := '"Type": "Template", "URI": "ST_BA_GeneralSettings"'}
	{attribute 'Description' := '"LCID": "1031", "Text": "Gebäude Wetterdaten"'}
	{attribute 'Description' := '"LCID": "1033", "Text": "Building Weather data"'}
{endregion}
FUNCTION_BLOCK FB_BA_WeatherData EXTENDS FB_BA_View
VAR_INPUT CONSTANT
	WthParam				: FB_BA_WeatherParameter;	
END_VAR
VAR // added by the converter: edge detectors and wires of the graphical bodies
    _s1 : ST_BA_GeneralSettings;
END_VAR

SUPER^(); // FB_BA_View
WthParam(fTWth := Site.stWeatherStation.fOutsideTemperature); // FB_BA_WeatherParameter
// compose _s1 : ST_BA_GeneralSettings
_s1.fFrostProtectionSetpoint := WthParam.fSpFrstProtec;
_s1.fTWthLowLimit := WthParam.fTWthLowLimit;
_s1.bTWthLowLimit := WthParam.bTWthLowLimit;
_s1.fTWthDamped := WthParam.fTWthDamped;
_s1.bTWthDampedLowLimit := WthParam.bTWthDampedLowLimit;
_s1.fTWth := Site.stWeatherStation.fOutsideTemperature;
Site.stGeneralSettings := _s1;

METHOD FB_init : BOOL
VAR_INPUT
	bInitRetains : BOOL; // if TRUE, the retain variables are initialized (warm start / cold start)
	bInCopyCode : BOOL;  // if TRUE, the instance afterwards gets moved into the copy code (online change)
END_VAR
WthParam.iParent			:= THIS^;
WthParam.iLabel				:= LblCtl_WeatherParameters;
WthParam.eDPADMode			:= E_BA_DPADMode.eInclude;
END_METHOD

END_FUNCTION_BLOCK

// ---- Templates/POUs/Trade/BuildingAutomation/Weather_Data/Parameter/FB_BA_WeatherParameter.TcPOU
{region '#Template'}
	{attribute 'Version' := '5.0.0.0'}
	{attribute 'Tags' := '"LCID": "1031", "Text": "General, Settings, Parameters, Basics"'}
	{attribute 'Tags' := '"LCID": "1033", "Text": "General, Settings, Parameters, Basics"'}
	{attribute 'Using' := '"Type": "Template", "URI": "BA2_Param"'}
	{attribute 'Description' := '"LCID": "1031", "Text": "Witterungsparameter für die Templates"'}
	{attribute 'Description' := '"LCID": "1033", "Text": "Weather parameters for the templates"'}
{endregion}
FUNCTION_BLOCK FB_BA_WeatherParameter EXTENDS FB_BA_View
VAR_INPUT
	fTWth					: REAL;	//	Weather temperature
END_VAR
VAR_OUTPUT
	fSpFrstProtec			: REAL;  // frost protection setpoint. for eg. Heating circutis in protection mode
	fTWthLowLimit			: REAL;  // below this value all frostprotection funcktions in HVAC-Plants will be enabled
	bTWthLowLimit			: BOOL;  // is TRUE when the outside temperature is below the value from fTWthLowLimit 
	fTWthDamped				: REAL;  // damped outside temperature
	bTWthDampedLowLimit		: BOOL;	
END_VAR
VAR_INPUT CONSTANT
	SpFrstProtec			: FB_BA_AV_Op;		
	TWthLowLimitVal			: FB_BA_AV_Op;																
	TWthLowLimit			: FB_BA_BV_Op;								
	TWthDamped				: FB_BA_AV_Op;		
	TWthDampedLowLimit		: FB_BA_BV_Op;	
END_VAR
VAR
	TWthLowLimitHys			: FB_BA_Swi2P;
	Average					: FB_BA_TiAvrg;
	TWthDampedLowLimitHys	: FB_BA_Swi2P;
END_VAR

SUPER^(); // FB_BA_View
SpFrstProtec(); // FB_BA_AV_Op
fSpFrstProtec := SpFrstProtec.fPresentValue;
TWthLowLimitVal(); // FB_BA_AV_Op
fTWthLowLimit := TWthLowLimitVal.fPresentValue;
TWthLowLimitHys(bEn := TRUE, fIn := fTWth, fOn := fTWthLowLimit, fOff := fTWthLowLimit + 1.0); // FB_BA_Swi2P
TWthLowLimit(bValuePgm := TWthLowLimitHys.bQ); // FB_BA_BV_Op
bTWthLowLimit := TWthLowLimit.bPresentValue;
Average(bEn := BA2_Param.bDlyStartPLC, fIn := fTWth, nIntval := 900, nNumOfElem := 96); // FB_BA_TiAvrg
TWthDamped(fValuePgm := Average.fOut); // FB_BA_AV_Op
fTWthDamped := TWthDamped.fPresentValue;
TWthDampedLowLimitHys(bEn := TRUE, fIn := fTWthDamped, fOn := fTWthLowLimit, fOff := fTWthLowLimit + 1.0); // FB_BA_Swi2P
TWthDampedLowLimit(bValuePgm := TWthDampedLowLimitHys.bQ); // FB_BA_BV_Op
bTWthDampedLowLimit := TWthDampedLowLimit.bPresentValue;

METHOD FB_init : BOOL
VAR_INPUT
	bInitRetains : BOOL; // if TRUE, the retain variables are initialized (warm start / cold start)
	bInCopyCode : BOOL;  // if TRUE, the instance afterwards gets moved into the copy code (online change)
END_VAR
SpFrstProtec.iParent				:= THIS^;
SpFrstProtec.iLabel					:= LblCtl_SetpointFrostProtection;
SpFrstProtec.eUnit					:= E_BA_Unit.eTemperature_DegreesCelsius;  
SpFrstProtec.fValueRm				:= 5.0;
SpFrstProtec.fCOVIncrement			:= BA2_Param.fDefCOVIncrement;							

TWthLowLimitVal.iParent				:= THIS^;
TWthLowLimitVal.iLabel				:= LblCtl_SetpointMinimumOutsideTemperature;
TWthLowLimitVal.eUnit				:= E_BA_Unit.eTemperature_DegreesCelsius;  
TWthLowLimitVal.fValueRm			:= 8.0;
TWthLowLimitVal.fCOVIncrement		:= BA2_Param.fDefCOVIncrement;							

TWthLowLimit.iParent				:= THIS^;	
TWthLowLimit.iLabel					:= LblCtl_OperationalMessageTemperatureWeatherLowLimit;
TWthLowLimit.sInactiveText			:= txtEvent_Off;
TWthLowLimit.sActiveText			:= txtEvent_On;
TWthLowLimit.bValueRm				:= FALSE;		
TWthLowLimit.eToggleMode 			:= E_BA_ToggleMode.eSwitch;

TWthDamped.iParent					:= THIS^;
TWthDamped.iLabel					:= LblCtl_MeanDamped;
TWthDamped.eUnit					:= E_BA_Unit.eTemperature_DegreesCelsius;  
TWthDamped.fValueRm					:= 0.0;
TWthDamped.fCOVIncrement			:= BA2_Param.fDefCOVIncrement;							

TWthDampedLowLimit.iParent			:= THIS^;	
TWthDampedLowLimit.iLabel			:= LblCtl_OperationalMessageTemperatureWeatherDampedLowLimit;	
TWthDampedLowLimit.sInactiveText	:= txtEvent_Off;
TWthDampedLowLimit.sActiveText		:= txtEvent_On;
TWthDampedLowLimit.bValueRm			:= FALSE;								
TWthDampedLowLimit.eToggleMode 		:= E_BA_ToggleMode.eSwitch;
END_METHOD

END_FUNCTION_BLOCK

// ---- Templates/POUs/Trade/HeatingSystem/FB_BA_Heating.TcPOU
{region '#Template'}
	{attribute 'Version' := '5.0.0.0'}
	{attribute 'Tags' := '"LCID": "1031", "Text": "Trade, Plant, Heating System"'}
	{attribute 'Tags' := '"LCID": "1033", "Text": "Trade, Plant, Heating System"'}
	{attribute 'Using' := '"Type": "Template", "URI": "Site"'}
	{attribute 'Description' := '"LCID": "1031", "Text": "Aufruf der Anlagen des Gewerks Heizsysteme"'}
	{attribute 'Description' := '"LCID": "1033", "Text": "Calling the plants of the trade heating system"'}
{endregion}
FUNCTION_BLOCK FB_BA_Heating EXTENDS FB_BA_View
VAR_INPUT CONSTANT
	HTC01				: FB_BA_H_HtgCir01;		
END_VAR
VAR_INPUT
END_VAR
VAR_OUTPUT
END_VAR
VAR
END_VAR

SUPER^(); // FB_BA_View
HTC01(); // FB_BA_H_HtgCir01

METHOD FB_init : BOOL
VAR_INPUT
	bInitRetains : BOOL; // if TRUE, the retain variables are initialized (warm start / cold start)
	bInCopyCode : BOOL;  // if TRUE, the instance afterwards gets moved into the copy code (online change)
END_VAR
HTC01.iParent 					:= THIS^;	
HTC01.iLabel					:= LblPlt_Heating_circuit;	
HTC01.sObjectName				:= '{Idx=01}';  
HTC01.eDPADMode					:= E_BA_DPADMode.eInclude;
END_METHOD

END_FUNCTION_BLOCK

// ---- Templates/POUs/Trade/HazardDetectionAlarmSystems/FB_BA_HazardDetectionAlarmSystems.TcPOU
{region '#Template'}
	{attribute 'Version' := '5.1.0.0'}
	{attribute 'Tags' := '"LCID": "1031", "Text": "Gebäudeautomation, Alarme"'}
	{attribute 'Tags' := '"LCID": "1033", "Text": "Building automation, Alarms"'}
	{attribute 'Description' := '"LCID": "1031", "Text": "Gebäude Alarme"'}
	{attribute 'Description' := '"LCID": "1033", "Text": "Building Alarms"'}
{endregion}
FUNCTION_BLOCK FB_BA_HazardDetectionAlarmSystems EXTENDS FB_BA_View
VAR_INPUT
END_VAR
VAR_OUTPUT
END_VAR
VAR_INPUT CONSTANT
	FireAlarmSystem01			: FB_BA_FireAlarmSystem;
	BurglarAlarmSystem01		: FB_BA_BurglarAlarmSystem;
END_VAR
VAR
END_VAR

SUPER^(); // FB_BA_View
FireAlarmSystem01(); // FB_BA_FireAlarmSystem
BurglarAlarmSystem01(); // FB_BA_BurglarAlarmSystem

METHOD FB_init : BOOL
VAR_INPUT
	bInitRetains : BOOL; // if TRUE, the retain variables are initialized (warm start / cold start)
	bInCopyCode : BOOL;  // if TRUE, the instance afterwards gets moved into the copy code (online change)
END_VAR
FireAlarmSystem01.iParent			:= THIS^;	
FireAlarmSystem01.iLabel			:= LblPlt_Fire_detection_and_alarm_systems;
FireAlarmSystem01.sObjectName		:= '{Idx=61}';
FireAlarmSystem01.eDPADMode			:= E_BA_DPADMode.eInclude;

BurglarAlarmSystem01.iParent		:= THIS^;	
BurglarAlarmSystem01.iLabel			:= LblPlt_Burglar_alarm_systems;
BurglarAlarmSystem01.sObjectName	:= '{Idx=71}';
BurglarAlarmSystem01.eDPADMode		:= E_BA_DPADMode.eInclude;
END_METHOD

END_FUNCTION_BLOCK

// ---- Templates/POUs/Trade/AutomationControl/Device/TimeSettings/FB_BA_ExternalSysTime.TcPOU
{region '#Template'}
	{attribute 'Version' := '5.0.1.0'}
	{attribute 'Tags' := '"LCID": "1031", "Text": "Automatisierungssteuerung, Gerät, Einstellungen, Systemzeit, BACnet Adapter Time"'}
	{attribute 'Tags' := '"LCID": "1033", "Text": "Automation control, Device, Settings, Systemzeit, BACnet Adapter Zeit"'}
	{attribute 'Using' := '"Type": "Template", "URI": "SysTime"'}		 		 
	{attribute 'Description' := '"LCID": "1031", "Text": "Externe Systemzeit abrufen und lokal setzen"'}
	{attribute 'Description' := '"LCID": "1033", "Text": "Get external system time and set locally"'}
{endregion}

FUNCTION_BLOCK FB_BA_ExternalSysTime
VAR_INPUT
END_VAR
VAR_OUTPUT
END_VAR
VAR_INPUT CONSTANT PERSISTENT	
	sExternalAmsNetId						: T_AmsNetId := ''; // Beispiel,Example: '192.168.131.1.1.1'
	{attribute 'parameterUnit':= 's'}
	GetExtSysTime_nTiAuto					: UDINT := 600;
	{attribute 'parameterUnit':= 's'}
	GetLocalSysTime_nTiAuto					: UDINT := 60;
END_VAR	
VAR_INPUT CONSTANT
	GetExtSysTime				: FB_BA_GetTime;

	SetSysTimeLocal				: FB_BA_SetTime;
	SetBACnetAdapterTime		: FB_BACnet_SetAdapterTime;

	GetLocalSysTime				: FB_BA_GetTime;
	GetBACnetAdapterTime		: FB_BACnet_GetAdapterTime;
END_VAR
VAR
	GetExtSysTime_bSync					: BOOL;	
	GetExtSysTime_rtrigSync				: R_TRIG;
	
